(* CoDeSys 2.3 project: cy-07-wg-004.pro *)
(* Title: ClevergyAS - Albino E-02 *)
(* Version: 1.25 *)
(* Author: Andrea Ravasio *)
(* Libraries: ModbusEthernet_03.lib 20.1.16 10:42:42, Standard.lib 2.12.10 14:48:34, Util.lib 26.9.14 10:12:46, Visual.lib 2.12.10 14:48:34, LON_01.lib 28.9.12 14:05:10, WagoLibIdent.lib 25.2.13 11:12:16, WagoLibMBX_01.lib 20.3.12 16:32:40, SysLibSockets.lib 10.2.11 09:20:54, Ethernet.lib 2.12.10 14:48:32, WagoLibStatus.lib 2.12.10 14:48:32, SysLibFile.lib 2.12.10 14:48:34, SysLibRtc.lib 2.12.10 14:48:32, SysLibEvent.lib 2.12.10 14:48:34, SysLibPlcCtrl.lib 2.12.10 14:48:32, SysLibCallback.lib 2.12.10 14:48:32, Application\WagoLibEthernet_01.lib 2.12.10 14:48:36 *)

(* PLC configuration (modules and I/O channels)
VPN_ST1 AT %IX24.0 [BOOLOnX_I] Ch_1 Digital input
LAMP_AL AT %QX16.0 [BOOLOnX_Q] Ch_1 Digital output
KEY_QE_ST1 AT %IX24.1 [BOOLOnX_I] Ch_2 Digital input
CIRD05a_EN AT %QX16.1 [BOOLOnX_Q] Ch_2 Digital output
CIRD05b_AL AT %IX24.2 [BOOLOnX_I] Ch_3 Digital input
CIRD04b_EN AT %QX16.2 [BOOLOnX_Q] Ch_3 Digital output
CIRD05b_ST AT %IX24.3 [BOOLOnX_I] Ch_4 Digital input
CIRD04a_EN AT %QX16.3 [BOOLOnX_Q] Ch_4 Digital output
CIRD05b_AUT AT %IX24.4 [BOOLOnX_I] Ch_5 Digital input
CIRD03b_EN AT %QX16.4 [BOOLOnX_Q] Ch_5 Digital output
CIRD05a_AL AT %IX24.5 [BOOLOnX_I] Ch_6 Digital input
CIRD03a_EN AT %QX16.5 [BOOLOnX_Q] Ch_6 Digital output
CIRD05a_ST AT %IX24.6 [BOOLOnX_I] Ch_7 Digital input
CIRD02b_EN AT %QX16.6 [BOOLOnX_Q] Ch_7 Digital output
CIRD05a_AUT AT %IX24.7 [BOOLOnX_I] Ch_8 Digital input
CIRD02a_EN AT %QX16.7 [BOOLOnX_Q] Ch_8 Digital output
CIRD04b_AL AT %IX24.8 [BOOLOnX_I] Ch_1 Digital input
CIRD01b_EN AT %QX16.8 [BOOLOnX_Q] Ch_1 Digital output
CIRD04b_ST AT %IX24.9 [BOOLOnX_I] Ch_2 Digital input
CIRD01a_EN AT %QX16.9 [BOOLOnX_Q] Ch_2 Digital output
CIRD04b_AUT AT %IX24.10 [BOOLOnX_I] Ch_3 Digital input
CIRD05b_EN AT %QX16.10 [BOOLOnX_Q] Ch_3 Digital output
CIRD04a_AL AT %IX24.11 [BOOLOnX_I] Ch_4 Digital input
AT %QX16.11 [BOOLOnX_Q] Ch_4 Digital output
CIRD04a_ST AT %IX24.12 [BOOLOnX_I] Ch_5 Digital input
AT %QX16.12 [BOOLOnX_Q] Ch_5 Digital output
CIRD04a_AUT AT %IX24.13 [BOOLOnX_I] Ch_6 Digital input
AT %QX16.13 [BOOLOnX_Q] Ch_6 Digital output
CIRD03b_AL AT %IX24.14 [BOOLOnX_I] Ch_7 Digital input
AT %QX16.14 [BOOLOnX_Q] Ch_7 Digital output
CIRD03b_ST AT %IX24.15 [BOOLOnX_I] Ch_8 Digital input
AT %QX16.15 [BOOLOnX_Q] Ch_8 Digital output
CIRD03b_AUT AT %IX25.0 [BOOLOnX_I] Ch_1 Digital input
CIRD02b_AL AT %IX25.1 [BOOLOnX_I] Ch_2 Digital input
CIRD03a_AL AT %IX25.2 [BOOLOnX_I] Ch_3 Digital input
CIRD02b_ST AT %IX25.3 [BOOLOnX_I] Ch_4 Digital input
CIRD03a_ST AT %IX25.4 [BOOLOnX_I] Ch_5 Digital input
CIRD02b_AUT AT %IX25.5 [BOOLOnX_I] Ch_6 Digital input
CIRD03a_AUT AT %IX25.6 [BOOLOnX_I] Ch_7 Digital input
CIRD02a_AL AT %IX25.7 [BOOLOnX_I] Ch_8 Digital input
CIRD02a_ST AT %IX25.8 [BOOLOnX_I] Ch_1 Digital input
CIRD01b_AUT AT %IX25.9 [BOOLOnX_I] Ch_2 Digital input
CIRD02a_AUT AT %IX25.10 [BOOLOnX_I] Ch_3 Digital input
CIRD01a_AL AT %IX25.11 [BOOLOnX_I] Ch_4 Digital input
CIRD01b_AL AT %IX25.12 [BOOLOnX_I] Ch_5 Digital input
CIRD01a_ST AT %IX25.13 [BOOLOnX_I] Ch_6 Digital input
CIRD01b_ST AT %IX25.14 [BOOLOnX_I] Ch_7 Digital input
CIRD01a_AUT AT %IX25.15 [BOOLOnX_I] Ch_8 Digital input
ALARM_PM AT %IX26.0 [BOOLOnX_I] Ch_1 Digital input
AT %IX26.1 [BOOLOnX_I] Ch_2 Digital input
ALARM_PB AT %IX26.2 [BOOLOnX_I] Ch_3 Digital input
AT %IX26.3 [BOOLOnX_I] Ch_4 Digital input
ALARM_TB AT %IX26.4 [BOOLOnX_I] Ch_5 Digital input
AT %IX26.5 [BOOLOnX_I] Ch_6 Digital input
CTL01_ST AT %IX26.6 [BOOLOnX_I] Ch_7 Digital input
AT %IX26.7 [BOOLOnX_I] Ch_8 Digital input
AT %IB0 [BYTEOnB_I] First Byte of 24
AT %QB0 [BYTEOnB_Q] First Byte of 24
0750-0464#04 2/4 AI RTD / ADJ./ HA [Type_44_4_Channels] node 6, in %IB48 out %QB28 {INTTypePAAssignment = PLC; INTTypeModule = plugged}
  T_S01 AT %IW12 [INTOnW_I] Ch_1 signed Input value
  T_S02 AT %IW13 [INTOnW_I] Ch_2 signed Input value
  T_S03 AT %IW14 [INTOnW_I] Ch_3 signed Input value
  T_S04 AT %IW15 [INTOnW_I] Ch_4 signed Input value
0750-0464#04 2/4 AI RTD / ADJ./ HA [Type_44_4_Channels] node 7, in %IB72 out %QB52 {INTTypePAAssignment = PLC; INTTypeModule = plugged}
  T_S07 AT %IW16 [INTOnW_I] Ch_1 signed Input value
  T_S06 AT %IW17 [INTOnW_I] Ch_2 signed Input value
  T_S05 AT %IW18 [INTOnW_I] Ch_3 signed Input value
  AT %IW19 [INTOnW_I] Ch_4 signed Input value
0750-0478 2 AI 0-10V 16 Bit S.E. [Type_8_2_Channels] node 8, in %IB80 out %QB52 {INTTypePAAssignment = PLC; INTTypeModule = plugged}
  VRD01_ST AT %IW20 [WORDOnW_I] Ch_1 Input word
  VRD02_ST AT %IW21 [WORDOnW_I] Ch_2 Input word
0750-0478 2 AI 0-10V 16 Bit S.E. [Type_8_2_Channels] node 9, in %IB88 out %QB52 {INTTypePAAssignment = PLC; INTTypeModule = plugged}
  VRD03_ST AT %IW22 [WORDOnW_I] Ch_1 Input word
  AT %IW23 [WORDOnW_I] Ch_2 Input word
0750-0556 2 AO ±10V [Type_14_2_Channels] node 10, in %IB92 out %QB52 {INTTypePAAssignment = PLC; INTTypeModule = plugged}
  VRD01_CTRL AT %QW12 [WORDOnW_Q] Ch_1 Analog output
  VRD02_CTRL AT %QW13 [WORDOnW_Q] Ch_2 Analog output
0750-0556 2 AO ±10V [Type_14_2_Channels] node 11, in %IB96 out %QB52 {INTTypePAAssignment = PLC; INTTypeModule = plugged}
  VRD03_CTRL AT %QW14 [WORDOnW_Q] Ch_1 Analog output
  AT %QW15 [WORDOnW_Q] Ch_2 Analog output
Fieldbus variables [FB_VARS] node 1, in %IB0 out %QB0
Flag variables [FLAG_VARS] node 2, in %IB0 out %QB0
Modbus-Master [MB_MASTER] node 3, in %IB0 out %QB0
*)

(* Global variable list: Addiitonal_Constants *)
VAR_GLOBAL CONSTANT

	Logger_MaxBCK : WORD:=100;

END_VAR

(* Global variable list: Additional_Retain *)
VAR_GLOBAL RETAIN PERSISTENT
	LogBCKIndex:  WORD;
END_VAR

(* Global variable list: Global_Constants *)
VAR_GLOBAL CONSTANT


	Plant_NAME			: STRING :='cySN:07 cyVER: E04 Palestra Palasport Albino ';
	Plant_SN			: DWORD  :=07(*07*);	(* S/N Impianto di telecontrollo *)
	Plant_SW_VER		: WORD   :=1;		(* Versione SW installata *)


	(* Colour defines *)
	COLOR_RED			: DWORD	:= 16#2020F0;
	COLOR_YELLOW		: DWORD	:= 16#20F0F0;
	COLOR_GREEN			: DWORD	:= 16#20F020;
	COLOR_LIGHT_GREEN	: DWORD := 16#006000;

	(* Parameters *)
	Plant_DefaultTAmb	: INT	:=100;		(* [.1°C] Temperatura ambiente di default in caso di rottura sonda *)
	Plant_MaxRunTAmb	: INT   :=210; 		(* [.1°C] Temperatura ambiente massima funzionamento impianto *)
	Plant_AntiFreezeTAmb: INT   :=-40;		(* [.1°C] Antifreeze temperature, start circulators *)
	Plant_VRD_TAlarm	: INT   :=850; 		(* [.1°C] Temperatura di allarme VRD, blocco *)
	Plant_VRD_TMax		: INT   :=800; 		(* [.1°C] Setpoint massimo per uscita VRD *)
	Plant_VRD_TDefault	: INT	:=300;		(* [.1°C] Temperatura di default in caso di errore climatica *)
	Plant_CirOffDelay	: TIME	:=T#30m;	(* (Def.T#15m) Ritardo spegnimento pompe per ricircolo caldaia *)
	Plant_CirOnDelay	: TIME	:=T#15m;
	Plant_MaxWaterLoss	: WORD  :=2;		(* [lt/h] Massima perdita del circuito *)

	(* Filesystem *)
	FilesPath  			: STRING :='S:\';

	(* TCP Logger *)
	Logger_SERVER		: STRING:='';
	Logger_IP			: STRING:='192.168.100.3';(*'178.33.227.41'; (*  *) *)
	Logger_PORT			: WORD  :=80;
	Logger_GETSTART		: STRING:='GET /cygmsrv/hsgm.ashx?';
	Logger_GETEND		: STRING:='$R$N$R$N';
	Logger_CHECK		: STRING:='True';
	Logger_CRLF			: STRING:='$R$N';
	Logger_DataFile		: STRING:='S:\LOG.DAT';
	Logger_DataFileOld	: STRING:='S:\LOG.BCK';
	Logger_IndexFile	: STRING:='S:\LOG.IDX';
	Logger_ConnRetries	: BYTE:=5;
	Logger_RecoverMsgs	: BYTE:=25;

	(* TCP Remote *)
	Remote_PORT			: WORD  :=10;
	Remote_WELCOME		: STRING:='Connected$R$N';
	Remote_OK			: STRING:='OK$R$N';
	Remote_ERROR		: STRING:='ERROR$R$N';

	(* TCP Sockets *)
	MAX_SEND_TCP_SERVER					 : DWORD:=3000;(*60000*)
	MAX_RECEIVE_TCP_SERVER				 : DWORD:=3000;
	MAX_RECEIVE_TCP_SERVER_SOCKET	 	 : DWORD:=1500;
	MAX_SEND_TCP_CLIENT					 : DWORD:=3000;(*15000*)
	MAX_RECEIVE_TCP_CLIENT				 : DWORD:=1500;
	MAX_RECEIVE_TCP_CLIENT_SOCKET		 : DWORD:=1500;
	MAX_RECEIVE_UDP_SERVER				 : INT  :=1472;
	MAX_RECEIVE_UDP_CLIENT				 : INT  :=1472;
	CONNECT_WATCHDOG_TIME				 : TIME :=t#10s;

END_VAR

(* Global variable list: Global_Retain *)
VAR_GLOBAL RETAIN PERSISTENT
	CAL01_Clima : typ_Clima;
	VRD01_Clima : typ_Clima;
	VRD02_Clima : typ_Clima;
	VRD03_Clima : typ_Clima;

	CTL01_Count : DWORD;

	Mode_Manual : BOOL := FALSE;



	DelayAllarmeTemperaturaNonRaggiunta: INT;
	DeltaInterventoAllarmeTempeaturaNonRaggiuta: INT;
	OffsetSetPointManuale:INT;							(* Offset al Setpoint manuale per comensare lo scambiatore *)

	SogliaMinStartAntigelo: INT;
	SogliaMinStopAntigelo: INT;
	BitAbilitaAntigelo: BOOL:=TRUE;

END_VAR

(* Global variable list: Global_Variables *)
VAR_GLOBAL

	SYS    : typ_SYS;
	Logger : typ_Logger;


(*	Lamp	:	PLANT_STATUS; *)
	Lamp	:	LAMP_AL_GENERALE;

	T_AMB	:	INT;		(* Environment temperature *)

	TPV01  : obj_TPV	:= ( ID:=1 ); 							   (* T_S01 *)
	TPV02  : obj_TPV	:= ( ID:=2 , IN_WMIN:=50 , IN_WMAX:=870, IN_EMAX:=900 ); (* T_S02 - CAL01 - T_Send *)
	TPV03  : obj_TPV	:= ( ID:=3 , IN_WMIN:=50 , IN_WMAX:=850, IN_EMAX:=900 ); (* T_S03 *)
	TPV04  : obj_TPV	:= ( ID:=4 , IN_WMIN:=50 , IN_WMAX:=800 ); (* T_S04 *)
	TPV05  : obj_TPV	:= ( ID:=5 , IN_WMIN:=50 , IN_WMAX:=800 ); (* T_S05 *)
	TPV06  : obj_TPV	:= ( ID:=6 , IN_WMIN:=50 , IN_WMAX:=800 ); (* T_S06 *)
	TPV07  : obj_TPV	:= ( ID:=7 , IN_WMIN:=50 , IN_WMAX:=800 ); (* T_S07 *)
	TPV08  : obj_TPV	:= ( ID:=8 , IN_WMIN:=50 , IN_WMAX:=800 ); (* T_S08 per Gestione SPLIT *)
	TPV09  : obj_TPV	:= ( ID:=9 , IN_WMIN:=50 , IN_WMAX:=800 ); (* T_S09 per Gestione SPLIT *)
	TPV10  : obj_TPV	:= ( ID:=10 , IN_WMIN:=50 , IN_WMAX:=800 ); (* T_S10 per Gestione SPLIT *)
	TPV11  : obj_TPV	:= ( ID:=11 , IN_WMIN:=50 , IN_WMAX:=800 ); (* T_S11 per Gestione SPLIT *)

	TAMB   : obj_TAMB	:= ( ID:=1 );

	CAL01  : obj_CAL_VT100GC1B := ( ID:=1 );

	THER01 : obj_CRONTER_01 := ( ID:=1, Local_MaxRunTAmb:=250,Histeresys:=10);  (* Controllo Split 10 e 11 *)
	THER02 : obj_CRONTER_01 := ( ID:=2, Local_MaxRunTAmb:=250,Histeresys:=10);	(* Controllo SPLIt 4,5 e 6 *)
	THER03 : obj_CRONTER_01 := ( ID:=3, Local_MaxRunTAmb:=250,Histeresys:=10);	(* Controllo Split 8,9 e 10 *)
	THER04 : obj_CRONTER_01 := ( ID:=4, Local_MaxRunTAmb:=250,Histeresys:=10);	(* Controllo SPLIt 1,2 e 3 *)
	THER05 : obj_CRONTER_01 := ( ID:=5, Local_MaxRunTAmb:=250,Histeresys:=10);	(* Controllo Circolatore CIRD05 Servizi *)
	THER06 : obj_CRONTER_01 := ( ID:=6, Local_MaxRunTAmb:=800,Histeresys:=10);	(* Controllo Circolatore CIRD02 Bollitore *)
	THER07 : obj_CRONTER_01 := ( ID:=7, Local_MaxRunTAmb:=250,Histeresys:=10);	(* Controllo Ciroclatore CIRD03 ACS *)
	THER250 : obj_CRONTER_01 := ( ID:=250 );	(* Controllo Boost *)

	CronEd : obj_CRON_EDITOR_01;

	(* Circolatori  *)
	CIRD01 :obj_CIR_DOPPIO_new := (ID:=1, OnDelay:=T#1m, ExtStatus:=FALSE, Mode:=1); (* Primario Caldaia *)
	CIRD02 :obj_CIR_DOPPIO_new := (ID:=2, OnDelay:=T#1m, ExtStatus:=FALSE, Mode:=0); (* Secondario Bollitore *)
	CIRD03 :obj_CIR_DOPPIO_new := (ID:=3, OnDelay:=T#1m, ExtStatus:=FALSE, Mode:=0); (* Secondario ACS *)
	CIRD04 :obj_CIR_DOPPIO_new := (ID:=4, OnDelay:=T#1m, ExtStatus:=FALSE, Mode:=0); (* Secondario Ariotermi *)
	CIRD05 :obj_CIR_DOPPIO_new := (ID:=5, OnDelay:=T#1m, ExtStatus:=FALSE, Mode:=0); (* Secondario Servizi *)



	(* Valvole motorizzate Analogiche  *)
	VRD01	:	obj_VRD_new	:= (ID:=1, fFeedback:=TRUE, ReducedRange := FALSE , Local_VRD_TAlarm:=800);
	VRD02	:	obj_VRD_new := (ID:=2, fFeedback:=TRUE, ReducedRange := FALSE , Local_VRD_TAlarm:=800);
	VRD03	:	obj_VRD_new := (ID:=3, fFeedback:=TRUE, ReducedRange := FALSE, Local_VRD_TAlarm:=800);

	CTL01	:	obj_CTL	:= (ID:=1, Peso:=100);  (**** 0,5 litri al minuto : 2 impulsi al litro ***)

	SPL01:obj_SPLIT:= ( ID:=1);
	SPL02:obj_SPLIT:= ( ID:=2);
	SPL03:obj_SPLIT:= ( ID:=3);
	SPL04:obj_SPLIT:= ( ID:=4);
	SPL05:obj_SPLIT:= ( ID:=5);
	SPL06:obj_SPLIT:= ( ID:=6);
	SPL07:obj_SPLIT:= ( ID:=7);
	SPL08:obj_SPLIT:= ( ID:=8);
	SPL09:obj_SPLIT:= ( ID:=9);
	SPL10:obj_SPLIT:= ( ID:=10);
	SPL11:obj_SPLIT:= ( ID:=11);


(* Variabili Globali letti dal remoto della Palestra *)

	KEY_QE_ST2: BOOL;
	SPLIT06_ST: BOOL;
	SPLIT08_ST: BOOL;
	SPLIT05_ST: BOOL;
	SPLIT07_ST: BOOL;
	SPLIT04_ST: BOOL;
	SPLIT01_ST: BOOL;
	SPLIT09_ST: BOOL;
	SPLIT02_ST: BOOL;
	SPLIT11_ST: BOOL;
	SPLIT03_ST: BOOL;
	SPLIT10_ST: BOOL;
	SPLIT06_EN: BOOL;
	SPLIT05_EN: BOOL;
	SPLIT04_EN: BOOL;
	SPLIT09_EN: BOOL;
	SPLIT08_EN: BOOL;
	SPLIT07_EN: BOOL;
	SPLIT01_EN: BOOL;
	SPLIT02_EN: BOOL;
	SPLIT03_EN: BOOL;
	SPLIT11_EN: BOOL;
	SPLIT10_EN: BOOL;


	T_S08:INT;
	T_S09:INT;
	T_S10:INT;
	T_S11:INT;







END_VAR

(* Global variable list: LON/Module_1/InterfaceBlock_Module_1 *)
VAR_GLOBAL CONSTANT
(******************************************)
(* Automatic generated code, do not edit! *)
(******************************************)
	abSignature_Module_1 : ARRAY[0..15] OF BYTE := 16#B4,16#A9,16#CB,16#FD,16#2D,16#5A,16#D7,16#4A,16#B1,16#7E,16#A8,16#70,16#0A,16#0F,16#B9,16#03;
	wConfigSize_Module_1 : WORD := 421;
	abInterface_Module_1 : ARRAY[0..105] OF DWORD :=
		16#50A640DC, 16#219F340B, 16#6041B800, 16#06246830, 16#428B2E71, 16#64B95263, 16#FE000902, 16#2A050140, 
		16#0028408B, 16#20280AF2, 16#80A205C4, 16#685174C0, 16#8E03020C, 16#B8AB63AE, 16#953A4EEA, 16#AA63AD8E, 
		16#63ACD182, 16#4EEB98AD, 16#313DBE3A, 16#A6020F80, 16#13011245, 16#9926B18A, 16#0994A6CB, 16#508D4E85, 
		16#F6AD5BAA, 16#C53E2D4B, 16#EED8B26A, 16#920DBA93, 16#DBBC20C9, 16#0529B7EE, 16#B66DDF8E, 16#49D76DD9, 
		16#72CBA205, 16#1626C0B2, 16#A5A6B5EB, 16#6CDDB865, 16#4CA03BB7, 16#8AC91726, 16#3BF5AD0C, 16#75E986A5, 
		16#E2C9A3B9, 16#5AA34208, 16#4054966D, 16#946ACAA7, 16#49264935, 16#23655360, 16#E3E92DD4, 16#1524C09B, 
		16#A97EA56A, 16#4E053D69, 16#C906C1CA, 16#54CA1922, 16#E586651B, 16#12B5706D, 16#D3AF5791, 16#A0FA824C, 
		16#D202B450, 16#D069007C, 16#A940D4E8, 16#EAC16D51, 16#83B21003, 16#8B579930, 16#79D912B9, 16#02ED1029, 
		16#DDB14145, 16#6D5B962A, 16#B7471BC0, 16#511C9520, 16#3D44BB68, 16#1BAC9C4E, 16#61E7861D, 16#A1D85F80, 
		16#823280B0, 16#B3FF0007, 16#6C109AC5, 16#30A13C03, 16#E2386308, 16#58DB08B0, 16#6F400DE6, 16#0701DA1C, 
		16#98F51C73, 16#40A0630F, 16#AEE3AF23, 16#632020C0, 16#402040AF, 16#1605B0E3, 16#185B0CC4, 16#EDC04D71, 
		16#0610584B, 16#001688C7, 16#4544F1F8, 16#1C1713C6, 16#71815C54, 16#CA454672, 16#0696150F, 16#120412D0, 
		16#4C973101, 16#44A16C67, 16#2820D488, 16#E04081E0, 16#2F4F4D9B, 16#75AD2DFB, 16#F61B5BE9, 16#870AE1A2, 
		16#1B7860EE, 16#00000090;
END_VAR

(* Global variable list: LON/Module_1/Runtime_Module_1 *)
VAR_GLOBAL
(******************************************)
(* Automatic generated code, do not edit! *)
(******************************************)
	mbxModule_1 : MBX_Full;
	InDataTelegram_Module_1 : ARRAY[0..255] OF BYTE;
	OutDataTelegram_Module_1 : ARRAY[0..511] OF BYTE;

	xInitRunning_Module_1 : BOOL := FALSE;
	unLastLen_mbxModule_1 : UINT;
END_VAR

(* Data type in LON/Enumerations *)
TYPE alarm_type_t :
(
	AL_HEADER := -13,
	AL_FOOTER := -12,
	AL_DEBUG := -11,
	AL_INFO := -10,
	AL_SYSTEM_INFO := -6,
	AL_VALUE_INVALID := -5,
	AL_CONSTANT := -4,
	AL_OFFLINE := -3,
	AL_UNKNOWN := -2,
	AL_NUL := -1,
	AL_NO_CONDITION := 0,
	AL_ALM_CONDITION := 1,
	AL_TOT_SVC_ALM_1 := 2,
	AL_TOT_SVC_ALM_2 := 3,
	AL_TOT_SVC_ALM_3 := 4,
	AL_LOW_LMT_CLR_1 := 5,
	AL_LOW_LMT_CLR_2 := 6,
	AL_HIGH_LMT_CLR_1 := 7,
	AL_HIGH_LMT_CLR_2 := 8,
	AL_LOW_LMT_ALM_1 := 9,
	AL_LOW_LMT_ALM_2 := 10,
	AL_HIGH_LMT_ALM_1 := 11,
	AL_HIGH_LMT_ALM_2 := 12,
	AL_FIR_ALM := 13,
	AL_FIR_PRE_ALM := 14,
	AL_FIR_TRBL := 15,
	AL_FIR_SUPV := 16,
	AL_FIR_TEST_ALM := 17,
	AL_FIR_TEST_PRE_ALM := 18,
	AL_FIR_ENVCOMP_MAX := 19,
	AL_FIR_MONITOR_COND := 20,
	AL_FIR_MAINT_ALERT := 21,
	AL_FATAL_ERROR := 30,
	AL_ERROR := 31,
	AL_WARNING := 32
);
END_TYPE

(* Data type in Errors *)
TYPE en_Logger_ErrLev :
(
	EL_Log			:=0,
	EL_Wrn			:=1,
	EL_Alarm		:=2,
	EL_AlarmStop	:=3
);
END_TYPE

(* Data type in Errors *)
TYPE en_Logger_Status :
(
	S_Logger_UNKNOWN := 0,
	S_Logger_IDLE,
	S_Logger_WAITCONN,
	S_Logger_WAITTX,
	S_Logger_WAITRESP,
	S_Logger_ERROR
);
END_TYPE

(* Data type *)
TYPE en_SYS_Objects :
(
	EO_SYS		:=0,  (* PLC *)
	EO_VPN		:=1,  (* VPN *)
	EO_DOOR		:=2,  (* Door & access control *)

	EO_CAL		:=10, (* Caldaia *)
	EO_CIR		:=11, (* Circolatore *)
	EO_CRON		:=12, (* Crono-termostato *)
	EO_VRD		:=13, (* Valvola miscelatore pannelli *)
	EO_CTL		:=14, (* Contalitri *)
	EO_CTB		:=15, (* Contabilizzatore *)
	EO_TPV		:=16, (* Temperature probes values *)
	EO_PPV		:=17, (* Pressure probes values *)
	EO_PBV		:=18, (* Over-Pressure Alarms *)
	EO_TBV		:=19, (* Over-Temperature Alarms *)
	EO_PMV		:=20, (* Under-Pressure Alarms *)
	EO_GRU		:=21, (* Gruppo termico *)
	EO_PDC		:=22, (* Pompa di calore *)
	EO_SOL		:=23, (* Pannello solare termico *)
	EO_ESOL		:=24, (* Pannello solare fotovoltaico *)
	EO_GAS		:=25, (* Contatore GAS *)
	EO_PORT		:=26, (* Misuratore di portata *)
	EO_FPV		:=27, (* Flow probes values *)
	EO_ANZ		:=28, (* Analizzatore di rete *)
	EO_SCA		:=29, (* Signal Control Alarms *)
	EO_LUX		:=30, (* Base Illumination point *)
	EO_LUXM		:=31, (* Metered Illumination point *)
	EO_PSG		:=32, (* Sensore di passaggio *)
	EO_HVAC		:=33, (* Heating, Ventilating and Air Conditioning *)
	EO_HYGRV	:=34, (* Relative Humidity sensors value *)
	EO_COOV		:=35, (* Carbon Dioxide CO2 sensors value *)
	EO_INV		:=36, (* Inverter *)
	EO_STR		:=37, (* Smart string box *)

	EO_SPT		:=38, (* SPLIT *)

	EO_CIRD		:=39, (* Double CIR *)
	EO_ACS		:=40, (* Hot domestic water *)
	EO_FRG		:=41, (* Frigo *)
	EO_THER		:=42, (* Thermostat *)
	EO_CIRM		:=43, (* Modbus CIR *)
	EO_CIRDM	:=44, (* Modbus double CIR *)

	EO_ZGW			:=200,  (* ZigBee - Gateway *)
	EO_ZRM			:=201,	(* ZigBee - Repeater *)
	EO_ZREL			:=202,	(* ZigBee - Actuator rele *)
	EO_ZTHL			:=203,	(* ZigBee - Temperature Sensor *)

	EO_ASGW			:=250,	(* ASi - Gateway *)
	EO_ASCBI		:=251,	(* ASi - Input Board, Ciabatta *)

	EO_LON			:=1000, (* Bus - LON *)
	EO_MODBUS		:=1001, (* Bus - MODBUS *)
	EO_MBUS			:=1002, (* Bus - M-BUS *)
	EO_MODBUS_TCP	:=1003, (* Bus - MODBUS TCP *)

	EO_GENERIC		:=9000, (* Generic dataset *)
	EO_EXPO			:=9001 (* EXPO dataset *)
);
END_TYPE

(* Data type *)
TYPE en_SYS_Status :
(
	S_UNKNOWN  := 0,
	S_STARTUP,
	S_INIT_RTC,
	S_INIT_VAR,
	S_AUTOTEST,
	S_RUNNING,
	S_SHUTDOWN,
	S_HALT
);
END_TYPE

(* Data type in LON/Enumerations *)
TYPE file_request_t :
(
	FR_NUL := -1,
	FR_OPEN_TO_SEND := 0,
	FR_OPEN_TO_RECEIVE := 1,
	FR_CLOSE_FILE := 2,
	FR_CLOSE_DELETE_FILE := 3,
	FR_DIRECTORY_LOOKUP := 4,
	FR_OPEN_TO_SEND_RA := 5,
	FR_OPEN_TO_RECEIVE_RA := 6
);
END_TYPE

(* Data type in LON/Enumerations *)
TYPE file_status_t :
(
	FS_NUL := -1,
	FS_XFER_OK := 0,
	FS_LOOKUP_OK := 1,
	FS_OPEN_FAIL := 2,
	FS_LOOKUP_ERR := 3,
	FS_XFER_UNDERWAY := 4,
	FS_IO_ERR := 5,
	FS_TIMEOUT_ERR := 6,
	FS_WINDOW_ERR := 7,
	FS_AUTH_ERR := 8,
	FS_ACCESS_UNAVAIL := 9,
	FS_SEEK_INVALID := 10,
	FS_SEEK_WAIT := 11
);
END_TYPE

(* Data type in LON/Enumerations *)
TYPE hvac_t :
(
	HVAC_NUL := -1,
	HVAC_AUTO := 0,
	HVAC_HEAT := 1,
	HVAC_MRNG_WRMUP := 2,
	HVAC_COOL := 3,
	HVAC_NIGHT_PURGE := 4,
	HVAC_PRE_COOL := 5,
	HVAC_OFF := 6,
	HVAC_TEST := 7,
	HVAC_EMERG_HEAT := 8,
	HVAC_FAN_ONLY := 9,
	HVAC_FREE_COOL := 10,
	HVAC_ICE := 11,
	HVAC_MAX_HEAT := 12,
	HVAC_ECONOMY := 13,
	HVAC_DEHUMID := 14,
	HVAC_CALIBRATE := 15,
	HVAC_EMERG_COOL := 16,
	HVAC_EMERG_STEAM := 17,
	HVAC_MAX_COOL := 18,
	HVAC_HVC_LOAD := 19,
	HVAC_NO_LOAD := 20
);
END_TYPE

(* Data type in LON/Enumerations *)
TYPE object_request_t :
(
	RQ_NUL := -1,
	RQ_NORMAL := 0,
	RQ_DISABLED := 1,
	RQ_UPDATE_STATUS := 2,
	RQ_SELF_TEST := 3,
	RQ_UPDATE_ALARM := 4,
	RQ_REPORT_MASK := 5,
	RQ_OVERRIDE := 6,
	RQ_ENABLE := 7,
	RQ_RMV_OVERRIDE := 8,
	RQ_CLEAR_STATUS := 9,
	RQ_CLEAR_ALARM := 10,
	RQ_ALARM_NOTIFY_ENABLED := 11,
	RQ_ALARM_NOTIFY_DISABLED := 12,
	RQ_MANUAL_CTRL := 13,
	RQ_REMOTE_CTRL := 14,
	RQ_PROGRAM := 15,
	RQ_CLEAR_RESET := 16,
	RQ_RESET := 17,
	RQ_CLEAR_LOG := 18,
	RQ_LOAD_PROGRAM := 19,
	RQ_RUN_PROGRAM := 20,
	RQ_HALT_PROGRAM := 21,
	RQ_RESTART_PROGRAM := 22,
	RQ_UNLOAD_PROGRAM := 23,
	RQ_STEP_PROGRAM := 24
);
END_TYPE

(* Data type in LON/Enumerations *)
TYPE priority_level_t :
(
	PR_NUL := -1,
	PR_LEVEL_0 := 0,
	PR_LEVEL_1 := 1,
	PR_LEVEL_2 := 2,
	PR_LEVEL_3 := 3,
	PR_1 := 4,
	PR_2 := 5,
	PR_3 := 6,
	PR_4 := 7,
	PR_6 := 8,
	PR_8 := 9,
	PR_10 := 10,
	PR_16 := 11
);
END_TYPE

(* Data type in Plant_Objects *)
TYPE typ_Clima : (* CURVA CLIMATICA *)
STRUCT
	InitOK:		BOOL;
	Points: 	ARRAY [0..10] OF POINT;
END_STRUCT
END_TYPE

(* Data type in Plant_Objects *)
TYPE typ_Cron_Calendar :
STRUCT
	Profile		: ARRAY[0..384] OF BYTE;
END_STRUCT
END_TYPE

(* Data type in Plant_Objects *)
TYPE typ_Cron_Jolly :
STRUCT
	Start		: DT;
	End			: DT;
	Temp		: WORD;
	Flags		: WORD; (* B0:Enabled B1..B15:Unused *)
END_STRUCT
END_TYPE

(* Data type in Plant_Objects *)
TYPE typ_Cron_Profile :
STRUCT
	Flags		: WORD;
	Setpoint	: ARRAY [0..95] OF WORD;
END_STRUCT
END_TYPE

(* Data type in Errors *)
TYPE typ_Logger :
STRUCT
	Status		: en_Logger_Status;

	SendReq		: BOOL;
	SendIdx		: DWORD;
	SendData	: ARRAY [0..MAX_SEND_TCP_CLIENT] OF BYTE;
	SendLen		: DINT;

	TData		: ARRAY [0..MAX_SEND_TCP_CLIENT] OF BYTE;
	TLen		: DINT;

	LastIdxPos	: DWORD;

	(* Temporary variables used by objects *)
	s1			: STRING(256);
	i1			: WORD;

END_STRUCT
END_TYPE

(* Data type in Plant_Objects *)
TYPE typ_MODBUS_VAR : (* Gestione parametri MODBUS *)
STRUCT
	SlaveAddress	: BYTE;
	FunCode			: BYTE;
	FunAddress		: WORD;
	Refresh_Time	: BYTE; (* 0:No refresh x:Refresh in seconds *)
	Refresh_Cnt		: BYTE; (* INTERNAL *)
	Variable		: POINTER TO WORD;
	Variable_Size	: BYTE;
	Variable_Mirror : WORD; (* INTERNAL [Force refresh on read variables when <>0] *)
END_STRUCT
END_TYPE

(* Data type *)
TYPE typ_SYS :
STRUCT
	Status			: en_SYS_Status;
	Warning			: BOOL;
	Alarm			: BOOL;
	AlarmStop		: BOOL;

	Time_LogString	: STRING;
	Time_Year		: WORD;
	Time_Month		: BYTE;
	Time_Day		: BYTE;
	Time_Hour		: BYTE;
	Time_Minute		: BYTE;

	Time_CT_DT		: DT;
	Time_CT_Day		: WORD;
	Time_CT_Quarter	: BYTE;

	LastLogs_Idx	: BYTE;
	LastLogs_Dat	: ARRAY[0..5] OF STRING;
	LastLogs_Msg	: ARRAY[0..5] OF STRING;

END_STRUCT
END_TYPE

(* Data type in LON/NetworkVariables *)
TYPE typSnvtAlarm : 
STRUCT
	abLocation : ARRAY[0..5] OF BYTE;
	wObjectId : WORD;
	bAlarmType : BYTE (* enum type alarm_type_t *);
	bPriorityLevel : BYTE (* enum type priority_level_t *);
	wIndexToSnvt : WORD;
	abValue : ARRAY[0..3] OF BYTE;
	wYear : WORD;
	bMonth : BYTE;
	bDay : BYTE;
	bHour : BYTE;
	bMinute : BYTE;
	bSecond : BYTE;
	wMillisecond : WORD;
	abAlarmLimit : ARRAY[0..3] OF BYTE;
	bStatusInformation : BYTE; (* bit allocation of bStatusInformation:
	bit 0: NVI update counter LSB
	bit 1: NVI update counter
	bit 2: NVI update counter
	bit 3: NVI update counter MSB
	bit 4: timeout for NVI occurs (MaxRcvTime expired)
	bit 5: reserved
	bit 6: reserved
	bit 7: force NVO update *)
	bInternalUseOnly : BYTE; (* Do not use this byte in your application! *)
END_STRUCT
END_TYPE

(* Data type in LON/NetworkVariables *)
TYPE typSnvtFilePos : 
STRUCT
	diRwPtr : DINT;
	wRwLength : WORD;
	bStatusInformation : BYTE; (* bit allocation of bStatusInformation:
	bit 0: NVI update counter LSB
	bit 1: NVI update counter
	bit 2: NVI update counter
	bit 3: NVI update counter MSB
	bit 4: timeout for NVI occurs (MaxRcvTime expired)
	bit 5: reserved
	bit 6: reserved
	bit 7: force NVO update *)
	bInternalUseOnly : BYTE; (* Do not use this byte in your application! *)
END_STRUCT
END_TYPE

(* Data type in LON/NetworkVariables *)
TYPE typSnvtFileReq : 
STRUCT
	bRequest : BYTE (* enum type file_request_t *);
	wIndex : WORD;
	wReceiveTimeout : WORD;
	abDestAddress : ARRAY[0..4] OF BYTE (* union declaration *);
	bAuthOn : BYTE;
	bPrioOn : BYTE;
	bStatusInformation : BYTE; (* bit allocation of bStatusInformation:
	bit 0: NVI update counter LSB
	bit 1: NVI update counter
	bit 2: NVI update counter
	bit 3: NVI update counter MSB
	bit 4: timeout for NVI occurs (MaxRcvTime expired)
	bit 5: reserved
	bit 6: reserved
	bit 7: force NVO update *)
	bInternalUseOnly : BYTE; (* Do not use this byte in your application! *)
END_STRUCT
END_TYPE

(* Data type in LON/NetworkVariables *)
TYPE typSnvtFileStatus : 
STRUCT
	bStatus : BYTE (* enum type file_status_t *);
	wNumberOfFiles : WORD;
	wSelectedFile : WORD;
	abAdr : ARRAY[0..21] OF BYTE (* union declaration *);
	bStatusInformation : BYTE; (* bit allocation of bStatusInformation:
	bit 0: NVI update counter LSB
	bit 1: NVI update counter
	bit 2: NVI update counter
	bit 3: NVI update counter MSB
	bit 4: timeout for NVI occurs (MaxRcvTime expired)
	bit 5: reserved
	bit 6: reserved
	bit 7: force NVO update *)
	bInternalUseOnly : BYTE; (* Do not use this byte in your application! *)
END_STRUCT
END_TYPE

(* Data type in LON/NetworkVariables *)
TYPE typSnvtHvacMode : 
STRUCT
	bSnvtHvacMode : BYTE (* enum type hvac_t *);
	bStatusInformation : BYTE; (* bit allocation of bStatusInformation:
	bit 0: NVI update counter LSB
	bit 1: NVI update counter
	bit 2: NVI update counter
	bit 3: NVI update counter MSB
	bit 4: timeout for NVI occurs (MaxRcvTime expired)
	bit 5: reserved
	bit 6: reserved
	bit 7: force NVO update *)
	bInternalUseOnly : BYTE; (* Do not use this byte in your application! *)
END_STRUCT
END_TYPE

(* Data type in LON/NetworkVariables *)
TYPE typSnvtObjRequest : 
STRUCT
	wObjectId : WORD;
	bObjectRequest : BYTE (* enum type object_request_t *);
	bStatusInformation : BYTE; (* bit allocation of bStatusInformation:
	bit 0: NVI update counter LSB
	bit 1: NVI update counter
	bit 2: NVI update counter
	bit 3: NVI update counter MSB
	bit 4: timeout for NVI occurs (MaxRcvTime expired)
	bit 5: reserved
	bit 6: reserved
	bit 7: force NVO update *)
	bInternalUseOnly : BYTE; (* Do not use this byte in your application! *)
END_STRUCT
END_TYPE

(* Data type in LON/NetworkVariables *)
TYPE typSnvtObjStatus : 
STRUCT
	wObjectId : WORD;
	bBitfieldByteOffset2 : BYTE (* bit field *);
	bBitfieldByteOffset3 : BYTE (* bit field *);
	bBitfieldByteOffset4 : BYTE (* bit field *);
	bBitfieldByteOffset5 : BYTE (* bit field *);
	bStatusInformation : BYTE; (* bit allocation of bStatusInformation:
	bit 0: NVI update counter LSB
	bit 1: NVI update counter
	bit 2: NVI update counter
	bit 3: NVI update counter MSB
	bit 4: timeout for NVI occurs (MaxRcvTime expired)
	bit 5: reserved
	bit 6: reserved
	bit 7: force NVO update *)
	bInternalUseOnly : BYTE; (* Do not use this byte in your application! *)
END_STRUCT
END_TYPE

(* Data type in LON/NetworkVariables *)
TYPE typSnvtState : 
STRUCT
	bBitfieldByteOffset0 : BYTE (* bit field *);
	bBitfieldByteOffset1 : BYTE (* bit field *);
	bStatusInformation : BYTE; (* bit allocation of bStatusInformation:
	bit 0: NVI update counter LSB
	bit 1: NVI update counter
	bit 2: NVI update counter
	bit 3: NVI update counter MSB
	bit 4: timeout for NVI occurs (MaxRcvTime expired)
	bit 5: reserved
	bit 6: reserved
	bit 7: force NVO update *)
	bInternalUseOnly : BYTE; (* Do not use this byte in your application! *)
END_STRUCT
END_TYPE

(* Data type in LON/NetworkVariables *)
TYPE typSnvtSwitch : 
STRUCT
	bValue : BYTE;
	siState : SINT;
	bStatusInformation : BYTE; (* bit allocation of bStatusInformation:
	bit 0: NVI update counter LSB
	bit 1: NVI update counter
	bit 2: NVI update counter
	bit 3: NVI update counter MSB
	bit 4: timeout for NVI occurs (MaxRcvTime expired)
	bit 5: reserved
	bit 6: reserved
	bit 7: force NVO update *)
	bInternalUseOnly : BYTE; (* Do not use this byte in your application! *)
END_STRUCT
END_TYPE

(* Data type in LON/NetworkVariables *)
TYPE typSnvtTempP : 
STRUCT
	iSnvtTempP : INT;
	bStatusInformation : BYTE; (* bit allocation of bStatusInformation:
	bit 0: NVI update counter LSB
	bit 1: NVI update counter
	bit 2: NVI update counter
	bit 3: NVI update counter MSB
	bit 4: timeout for NVI occurs (MaxRcvTime expired)
	bit 5: reserved
	bit 6: reserved
	bit 7: force NVO update *)
	bInternalUseOnly : BYTE; (* Do not use this byte in your application! *)
END_STRUCT
END_TYPE

(* Data type in LON/NetworkVariables *)
TYPE typSnvtTimeStamp : 
STRUCT
	iYear : INT;
	bMonth : BYTE;
	bDay : BYTE;
	bHour : BYTE;
	bMinute : BYTE;
	bSecond : BYTE;
	bStatusInformation : BYTE; (* bit allocation of bStatusInformation:
	bit 0: NVI update counter LSB
	bit 1: NVI update counter
	bit 2: NVI update counter
	bit 3: NVI update counter MSB
	bit 4: timeout for NVI occurs (MaxRcvTime expired)
	bit 5: reserved
	bit 6: reserved
	bit 7: force NVO update *)
	bInternalUseOnly : BYTE; (* Do not use this byte in your application! *)
END_STRUCT
END_TYPE

(* POU PLC_PRG, ST *)
PROGRAM PLC_PRG
VAR
	Timer1: TON; (* Fast controls tick *)
	Timer2: TON; (* Plant control tick *)
	Timer3: TON; (* Logger timer *)

(* Comunizaione con nodo WAGO 192.168.100.4 *)


	Master_1				:	ETHERNET_MODBUSMASTER_UDP;
	Funktion				:	BYTE := 16#17; 				(* READ_WRITE_REGISTERS *)

	ReadAddress				:	WORD := 16#0000;			(* Startadresse 		*)
	ReadQuantity			:	WORD := 16#0005;			(* Anzahl der Worte 	*)
	Rec_Buffer				:	ARRAY[1..255] OF WORD;	(* Empfangsdaten 	*)

	WriteAddress			:	WORD := 16#0000;			(* Startadresse		*)
	WriteQuantity			:	WORD := 16#0001;			(* Anzahl der Worte	*)
	Send_Buffer			:	ARRAY[1..255] OF WORD;	(* Sendedaten			*)

	Fehler					:	WORD;
	Fertig					:	BOOL;
	T1						:	TON;
	Z1						:	CTU;

	WordAppoggio: WORD;
	DelayAvvioCollegamentoWAGO: TON;
	HMI_AggiornaLog: BOOL;
	DelayAggiornamento: TON;
	TrigR_THER01: F_TRIG;
	VarApp: INT;
END_VAR



VAR_INPUT
	WriteOUT: WORD;
END_VAR

VAR_OUTPUT
	ReadWord: WORD;
END_VAR
(******************************************************************************
 ****                           MAIN TASK CODE                             ****
 ******************************************************************************

	Network setup:
		IP  = 192.168.100.2 | MSK = 255.255.255.0
		GW	= 192.168.100.1 | DNS = 192.168.100.1
		SNTP = 193.204.114.232 (3600s) ==> 192.168.100.3
*)

(*==============================*)
(*===== Main status machine ====*)
(*==============================*)
Main_Stm();



WordAppoggio.0:=SPLIT07_EN;
WordAppoggio.1:=SPLIT08_EN;
WordAppoggio.2:=SPLIT09_EN;
WordAppoggio.3:=SPLIT03_EN;
WordAppoggio.4:=SPLIT02_EN;
WordAppoggio.5:=SPLIT01_EN;
WordAppoggio.6:=SPLIT06_EN;
WordAppoggio.7:=SPLIT05_EN;
WordAppoggio.8:=SPLIT04_EN;
WordAppoggio.9:=SPLIT10_EN;
WordAppoggio.10:=SPLIT11_EN;
WriteOUT:=WordAppoggio;

DelayAvvioCollegamentoWAGO(IN:=TRUE , PT:=t#10s , Q=> , ET=> );
(* Provo a ritardare la lettura del nodo per veririfcare se il download del programma è più veloce *)
DelayAggiornamento(IN:=NOT DelayAggiornamento.Q,pt:=t#1s);

Fertig:=DelayAvvioCollegamentoWAGO.Q AND DelayAggiornamento.Q;

NodoWAGO();

KEY_QE_ST2:=ReadWord.0;
SPLIT03_ST:=ReadWord.1;
SPLIT07_ST:=ReadWord.2;
SPLIT02_ST:=ReadWord.3;
SPLIT08_ST:=ReadWord.4;
SPLIT01_ST:=ReadWord.5;
SPLIT09_ST:=ReadWord.6;
SPLIT06_ST:=ReadWord.7;
SPLIT05_ST:=ReadWord.8;
SPLIT10_ST:=ReadWord.9;
SPLIT04_ST:=ReadWord.10;
SPLIT11_ST:=ReadWord.11;



(*==============================*)
(*== Running cycle operations ==*)
(*==============================*)
IF SYS.Status>S_INIT_VAR THEN

	(* Update LON output variables (needs to be here to obtain only one refresh) *)
	CAL01.Heartbeat( CLIM:=CAL01_Clima );

	(* Execute LON process *)
	Module_1_PRG();

	(* Count water pulses *)
	CTL01(CTL_ST:=CTL01_ST, COUNT:=CTL01_Count);

			CIRD01(
					PumpA_AUTO:=CIRD01a_AUT,
					PumpB_AUTO:=CIRD01b_AUT ,
					PumpA_En=>CIRD01a_EN ,
					PumpB_EN=>CIRD01b_EN ,
					PumpA_AL:=NOT CIRD01a_AL,
					PumpB_AL:=NOT CIRD01b_AL,
					PumpA_ST:=CIRD01a_ST ,
					PumpB_ST:=CIRD01b_ST );

			CIRD02(
					PumpA_AUTO:=CIRD02a_AUT,
					PumpB_AUTO:=CIRD02b_AUT ,
					PumpA_En=>CIRD02a_EN ,
					PumpB_EN=>CIRD02b_EN ,
					PumpA_AL:=NOT CIRD02a_AL,
					PumpB_AL:=NOT CIRD02b_AL,
					PumpA_ST:=CIRD02a_ST ,
					PumpB_ST:=CIRD02b_ST );


			CIRD03(
					PumpA_AUTO:=CIRD03a_AUT,
					PumpB_AUTO:=CIRD03b_AUT ,
					PumpA_En=>CIRD03a_EN ,
					PumpB_EN=>CIRD03b_EN ,
					PumpA_AL:=NOT CIRD03a_AL,
					PumpB_AL:=NOT CIRD03b_AL,
					PumpA_ST:=CIRD03a_ST ,
					PumpB_ST:=CIRD03b_ST );

			CIRD04(
					PumpA_AUTO:=CIRD04a_AUT,
					PumpB_AUTO:=TRUE, (*CIRD04b_AUT , *)  (* questo ciroclatore è automatico *)
					PumpA_En=>CIRD04a_EN ,
					PumpB_EN=>CIRD04b_EN ,
					PumpA_AL:=NOT CIRD04a_AL,
					PumpB_AL:=NOT CIRD04b_AL,
					PumpA_ST:=CIRD04a_ST ,
					PumpB_ST:=CIRD04b_ST );

			CIRD05(
					PumpA_AUTO:=CIRD05a_AUT,
					PumpB_AUTO:=CIRD05b_AUT ,
					PumpA_En=>CIRD05a_EN ,
					PumpB_EN=>CIRD05b_EN ,
					PumpA_AL:=NOT CIRD05a_AL,
					PumpB_AL:=NOT CIRD05b_AL,
					PumpA_ST:=CIRD05a_ST ,
					PumpB_ST:=CIRD05b_ST );

(* SPLIT *)


			SPL01(	FeedBack_Contatore:=SPLIT01_ST ,SSPLIT_EN=> SPLIT01_EN );
			SPL02(	FeedBack_Contatore:=SPLIT02_ST ,SSPLIT_EN=> SPLIT02_EN );
			SPL03(	FeedBack_Contatore:=SPLIT03_ST ,SSPLIT_EN=> SPLIT03_EN );

			SPL04(	FeedBack_Contatore:=SPLIT04_ST ,SSPLIT_EN=> SPLIT04_EN );
			SPL05(	FeedBack_Contatore:=SPLIT05_ST ,SSPLIT_EN=> SPLIT05_EN );
			SPL06(	FeedBack_Contatore:=SPLIT06_ST ,SSPLIT_EN=> SPLIT06_EN );

			SPL07(	FeedBack_Contatore:=SPLIT07_ST ,SSPLIT_EN=> SPLIT07_EN );
			SPL08(	FeedBack_Contatore:=SPLIT08_ST ,SSPLIT_EN=> SPLIT08_EN );
			SPL09(	FeedBack_Contatore:=SPLIT09_ST ,SSPLIT_EN=> SPLIT09_EN );

			SPL10(	FeedBack_Contatore:=SPLIT10_ST ,SSPLIT_EN=> SPLIT10_EN );
			SPL11(	FeedBack_Contatore:=SPLIT11_ST ,SSPLIT_EN=> SPLIT11_EN );



END_IF

(*==============================*)
(*== System cycle operations ===*)
(*==============================*)
(* Execute TCP processes *)
Logger_Proc();
Remote_Proc();
(* Update user led *)
USRLED_Update();
(* Execute Cron Editor commands *)
CronEd();


(* Environment temperature *)
IF NOT TPV01.ERR THEN T_AMB := T_S01;
ELSE T_AMB := Plant_DefaultTAmb;
END_IF
END_PROGRAM
ACTION Main_Stm:
CASE Sys.Status OF

	S_STARTUP:
		Sys.Status:=S_INIT_RTC;

	S_INIT_RTC:
		(* Check RTC and update from network *)
		RTC_Update();
		(* Check time *)
		IF Sys.Time_Year>2000 THEN
			Sys.Status:=S_INIT_VAR;
		END_IF

	S_INIT_VAR:
		LogEv(EL_Wrn,EO_SYS,0,1,CONCAT('System_startup_v',WORD_TO_STRING(Plant_SW_VER)));
		Sys.Status:=S_RUNNING;

	S_RUNNING:
		Timer1(IN:=NOT Timer1.Q,PT:=T#50ms);
		IF Timer1.Q THEN
			(* Update meters *)
			CTL01 ( CTL_ST:=CTL01_ST, COUNT:=CTL01_Count );
			(* Update system checks *)
			SYS_Proc();
		END_IF

		Timer2(IN:=NOT Timer2.Q,PT:=T#500ms);
		IF Timer2.Q THEN
			(* Read current date/time *)
			RTC_Update();
			(* Execute plant operations *)
			TPV01	 ( IN:=T_S01 );
			TPV02	 ( IN:=T_S02 );
			TPV03	 ( IN:=T_S03 );
			TPV04	 ( IN:=T_S04 );
			TPV05	 ( IN:=T_S05 );
			TPV06	 ( IN:=T_S06 );
			TPV07	 ( IN:=T_S07 );
			TPV08	 ( IN:=T_S08 );
			TPV09	 ( IN:=T_S09 );
			TPV10	 ( IN:=T_S10 );
			TPV11	 ( IN:=T_S11 );

			TAMB  ( IN1:=TPV01, IN2:=TPV01 );


			(* Crono Termnostati  *)
			THER01(Temperature:=TPV10.AVG);
			SPL10.Split_RUN:=SEL(TPV10.ERR,THER01.Run,THER01.RunCrono); (* Piano Palestrina Alto *)
			SPL11.Split_RUN:=SEL(TPV10.ERR,THER01.Run,THER01.RunCrono); (* Piano Palestrina Basso *)

			(* per questi SPLIT è previsto la partenza in alternata quindi scambio l'isteresi locale tutte le volte che il conto spegne *)

			TrigR_THER01(clk:=THER01.Run);
			IF TrigR_THER01.Q THEN
				VarApp:=SPL10.TempIsteresiLocale;
				SPL10.TempIsteresiLocale:=SPL11.TempIsteresiLocale;
				SPL11.TempIsteresiLocale:=VarApp;
			END_IF



			(* Sicurezze e comandi *)
		 	SPL10(TemperaturaRiferimento:=THER01.Temperature,TemperaturaSet:=THER01.SetPoint,LimiteIsteresi:=THER01.Histeresys,TemperaturaOK:=TPV05.AVG>SPL10.SogliaTemperaturaMandata);
	 		SPL11(TemperaturaRiferimento:=THER01.Temperature,TemperaturaSet:=THER01.SetPoint,LimiteIsteresi:=THER01.Histeresys,TemperaturaOK:=TPV05.AVG>SPL11.SogliaTemperaturaMandata);


			(* Crono Termnostati  *)
			THER02(Temperature:=TPV08.AVG);
			SPL04.Split_RUN:=SEL(TPV08.ERR,THER02.Run,THER02.RunCrono); (* Palestra Lato SX Alto *)
			SPL05.Split_RUN:=SEL(TPV08.ERR,THER02.Run,THER02.RunCrono); (* Palestra Lato SX Centro *)
			SPL06.Split_RUN:=SEL(TPV08.ERR,THER02.Run,THER02.RunCrono); (* Palestra Lato SX Basso *)

			(* Sicurezze e comandi *)
		 	SPL04(TemperaturaRiferimento:=THER02.Temperature,TemperaturaSet:=THER02.SetPoint,LimiteIsteresi:=THER02.Histeresys,TemperaturaOK:=TPV05.AVG>SPL04.SogliaTemperaturaMandata);
	 		SPL05(TemperaturaRiferimento:=THER02.Temperature,TemperaturaSet:=THER02.SetPoint,LimiteIsteresi:=THER02.Histeresys,TemperaturaOK:=TPV05.AVG>SPL05.SogliaTemperaturaMandata);
	 		SPL06(TemperaturaRiferimento:=THER02.Temperature,TemperaturaSet:=THER02.SetPoint,LimiteIsteresi:=THER02.Histeresys,TemperaturaOK:=TPV05.AVG>SPL06.SogliaTemperaturaMandata);

			(* Crono Termnostati  *)
			THER03(Temperature:=TPV09.AVG);
			SPL07.Split_RUN:=SEL(TPV09.ERR,THER03.Run,THER03.RunCrono); (* Palestra Lato DX Alto *)
			SPL08.Split_RUN:=SEL(TPV09.ERR,THER03.Run,THER03.RunCrono); (* Palestra Lato DX Centro *)
			SPL09.Split_RUN:=SEL(TPV09.ERR,THER03.Run,THER03.RunCrono); (* Palestra Lato DX Basso *)

			(* Sicurezze e comandi *)
		 	SPL07(TemperaturaRiferimento:=THER03.Temperature,TemperaturaSet:=THER03.SetPoint,LimiteIsteresi:=THER03.Histeresys,TemperaturaOK:=TPV05.AVG>SPL07.SogliaTemperaturaMandata);
	 		SPL08(TemperaturaRiferimento:=THER03.Temperature,TemperaturaSet:=THER03.SetPoint,LimiteIsteresi:=THER03.Histeresys,TemperaturaOK:=TPV05.AVG>SPL08.SogliaTemperaturaMandata);
	 		SPL09(TemperaturaRiferimento:=THER03.Temperature,TemperaturaSet:=THER03.SetPoint,LimiteIsteresi:=THER03.Histeresys,TemperaturaOK:=TPV05.AVG>SPL09.SogliaTemperaturaMandata);

			(* Crono Termnostati  *)
			THER04(Temperature:=TPV11.AVG);
			SPL01.Split_RUN:=SEL(TPV11.ERR,THER04.Run,THER04.RunCrono); (* Gradinata Lato SX *)
			SPL02.Split_RUN:=SEL(TPV11.ERR,THER04.Run,THER04.RunCrono); (* Gradinata Lato Centro *)
			SPL03.Split_RUN:=SEL(TPV11.ERR,THER04.Run,THER04.RunCrono); (* Gradinata Lato DX *)

			(* Sicurezze e comandi *)
		 	SPL01(TemperaturaRiferimento:=THER04.Temperature,TemperaturaSet:=THER04.SetPoint,LimiteIsteresi:=THER04.Histeresys,TemperaturaOK:=TPV05.AVG>SPL01.SogliaTemperaturaMandata);
	 		SPL02(TemperaturaRiferimento:=THER04.Temperature,TemperaturaSet:=THER04.SetPoint,LimiteIsteresi:=THER04.Histeresys,TemperaturaOK:=TPV05.AVG>SPL02.SogliaTemperaturaMandata);
	 		SPL03(TemperaturaRiferimento:=THER04.Temperature,TemperaturaSet:=THER04.SetPoint,LimiteIsteresi:=THER04.Histeresys,TemperaturaOK:=TPV05.AVG>SPL03.SogliaTemperaturaMandata);






		(* Ciroclatore  Assevito agli SPLIT *)
			(* comndato dai vari cronotermostati *)
			CIRD04.OnOff:=THER01.Run OR THER02.Run
							OR THER03.Run OR THER04.Run;
	(*		(* comandato dai vari crono *)
			CIRD04.OnOff:=THER01.RunCrono OR THER02.RunCrono
							OR THER03.RunCrono OR THER04.RunCrono; *)

			(* Crono  *)
			THER05();
			CIRD05.OnOff:=THER05.RunCrono; (* Servizi *)

			(* Crono Termnostati  *)
			THER06(Temperature:=TPV04.AVG);
			CIRD02.OnOff:=SEL(TPV06.ERR,THER06.Run,THER06.RunCrono); (* Bollitore *)

			(* Crono  *)
			THER07();
			CIRD03.OnOff:=THER07.RunCrono; (* Servizi *)

			(*  l'offset Boost viene fatto direttamente sulle cliamtiche delle VRD perchè nonesiste la curva cliamtica della caldaia *)
			VRD01(RUN:=TRUE,CLIM:=VRD01_Clima,OffsetBoost:=THER250.SetPoint, TEMP:=TPV07.AVG, STATUS:=VRD01_ST, OUT=>VRD01_CTRL);
			VRD02(RUN:=CIRD04.Run, CLIM:=VRD02_Clima,OffsetBoost:=THER250.SetPoint, TEMP:=TPV05.AVG, STATUS:=VRD02_ST, OUT=>VRD02_CTRL);
			VRD03(RUN:=CIRD05.Run, CLIM:=VRD03_Clima,OffsetBoost:=THER250.SetPoint, TEMP:=TPV06.AVG, STATUS:=VRD03_ST, OUT=>VRD03_CTRL);


			THER250();



			(* Ciroclatore Primario Caldaia *)
			CIRD01.OnOff:=( CIRD02.Ctrl_Run OR CIRD04.Ctrl_Run OR CIRD05.Ctrl_Run ) AND SYS.AlarmStop=FALSE;

			(* Caldaia in RUN *)

			CAL01.Run := CIRD01.OnOff;


			(* Set Point Caldaia *)
			CAL01.SetPointManuale:=CAL01.Curve_Temp - OffsetSetPointManuale + THER250.SetPoint;  	(* Temperatrura del Boost *)

			CAL01.SetPointManuale:=MAX(CAL01.SetPointManuale,SEL(CIRD02.OnOff,0,THER06.SetPoint + OffsetSetPointManuale));
			CAL01.SetPointManuale:=MAX(CAL01.SetPointManuale,SEL(VRD01.RUN,0,VRD01.Ctrl_SetPoint));
			CAL01.SetPointManuale:=MAX(CAL01.SetPointManuale,SEL(VRD02.RUN,0,VRD02.Ctrl_SetPoint));
			CAL01.SetPointManuale:=MAX(CAL01.SetPointManuale,SEL(VRD03.RUN,0,VRD03.Ctrl_SetPoint));

			CAL01(CLIM:=CAL01_Clima,AbilitaSetPointManuale:=TRUE);


			Lamp( Allarme:=	(CAL01.Status_Log=2) OR
  						  	CIRD01.Status_Log=2 OR
  						  	CIRD02.Status_Log=2 OR
  						  	CIRD03.Status_Log=2 OR
 						  	CIRD04.Status_Log=2 OR
						  	CIRD05.Status_Log=2 OR
							TPV01.Status_Log=2 OR
							TPV02.Status_Log=2 OR
							TPV03.Status_Log=2 OR
							TPV04.Status_Log=2 OR
							TPV05.Status_Log=2 OR
							TPV06.Status_Log=2 OR
							TPV07.Status_Log=2 OR
							TPV08.Status_Log=2 OR
							TPV09.Status_Log=2 OR
							TPV10.Status_Log=2 OR
							TPV11.Status_Log=2 OR
							THER01.Status_Log=2 OR
							THER02.Status_Log=2 OR
							THER03.Status_Log=2 OR
							THER04.Status_Log=2 OR
							THER250.Status_Log=2 OR
							VRD01.Status_Log=2 OR
							VRD02.Status_Log=2 OR
							VRD03.Status_Log=2 OR
							SPL01.Status_Log=2 OR
							SPL01.Status_Log=2 OR
							SPL02.Status_Log=2 OR
							SPL03.Status_Log=2 OR
							SPL04.Status_Log=2 OR
							SPL05.Status_Log=2 OR
							SPL06.Status_Log=2 OR
							SPL07.Status_Log=2 OR
							SPL08.Status_Log=2 OR
							SPL09.Status_Log=2 OR
							SPL10.Status_Log=2 OR
							SPL11.Status_Log=2
							,
							Warning:=	(CAL01.Status_Log=1) OR
  						  	CIRD01.Status_Log=1 OR
  						  	CIRD02.Status_Log=1 OR
  						  	CIRD03.Status_Log=1 OR
 						  	CIRD04.Status_Log=1 OR
						  	CIRD05.Status_Log=1 OR
							TPV01.Status_Log=1 OR
							TPV02.Status_Log=1 OR
							TPV03.Status_Log=1 OR
							TPV04.Status_Log=1 OR
							TPV05.Status_Log=1 OR
							TPV06.Status_Log=1 OR
							TPV07.Status_Log=1 OR
							TPV08.Status_Log=1 OR
							TPV09.Status_Log=1 OR
							TPV10.Status_Log=1 OR
							TPV11.Status_Log=1 OR
							THER01.Status_Log=1 OR
							THER02.Status_Log=1 OR
							THER03.Status_Log=1 OR
							THER04.Status_Log=1 OR
							THER250.Status_Log=1 OR
							VRD01.Status_Log=1 OR
							VRD02.Status_Log=1 OR
							VRD03.Status_Log=1 OR
							SPL01.Status_Log=1 OR
							SPL01.Status_Log=1 OR
							SPL02.Status_Log=1 OR
							SPL03.Status_Log=1 OR
							SPL04.Status_Log=1 OR
							SPL05.Status_Log=1 OR
							SPL06.Status_Log=1 OR
							SPL07.Status_Log=1 OR
							SPL08.Status_Log=1 OR
							SPL09.Status_Log=1 OR
							SPL10.Status_Log=1 OR
							SPL11.Status_Log=1
							,
							AllarmeLampada=>LAMP_AL
							);



		END_IF

		Timer3(IN:=NOT Timer3.Q,PT:=T#5m);
		IF Timer3.Q OR HMI_AggiornaLog THEN
			(* Trig logger *)
			LogTrig();
			(* Execute temporary CSV logger *)
			CSV_Log();
		END_IF

	S_SHUTDOWN:
		(* Stop caldaia *)
		(* Stop deviatori *)
		(* Aspetta 5 min prima di spegnere eventuali circolatori *)
		Sys.Status:=S_STARTUP;

	S_HALT:
		(* Aspetta uscita manuale *)
		Sys.Status:=S_STARTUP;


ELSE
	Sys.Status:=S_STARTUP;
END_CASE;
END_ACTION
ACTION NodoWAGO:
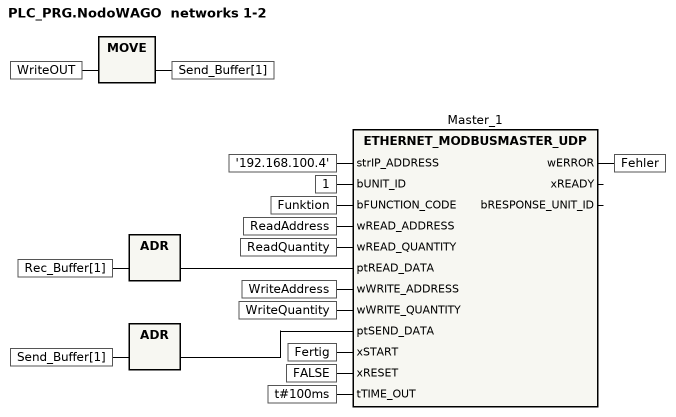
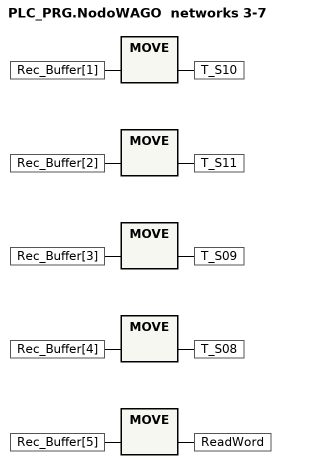
_FBD_ (* Function Block Diagram *)
NETWORK 1
	MOVE(WriteOUT) => Send_Buffer[1]
NETWORK 2
	Master_1:ETHERNET_MODBUSMASTER_UDP(strIP_ADDRESS: '192.168.100.4', bUNIT_ID: 1, bFUNCTION_CODE: Funktion, wREAD_ADDRESS: ReadAddress, wREAD_QUANTITY: ReadQuantity, ptREAD_DATA: ADR(Rec_Buffer[1]), wWRITE_ADDRESS: WriteAddress, wWRITE_QUANTITY: WriteQuantity, ptSEND_DATA: ADR(Send_Buffer[1]), xSTART: Fertig, xRESET: FALSE, tTIME_OUT: t#100ms) => Fehler
NETWORK 3
	MOVE(Rec_Buffer[1]) => T_S10
NETWORK 4
	MOVE(Rec_Buffer[2]) => T_S11
NETWORK 5
	MOVE(Rec_Buffer[3]) => T_S09
NETWORK 6
	MOVE(Rec_Buffer[4]) => T_S08
NETWORK 7
	MOVE(Rec_Buffer[5]) => ReadWord
_END_FBD_
(* the same logic as Structured Text *)
(* Network 1 *)
Send_Buffer[1] := WriteOUT;
(* Network 2 *)
Master_1(strIP_ADDRESS := '192.168.100.4', bUNIT_ID := 1, bFUNCTION_CODE := Funktion, wREAD_ADDRESS := ReadAddress, wREAD_QUANTITY := ReadQuantity, ptREAD_DATA := ADR(Rec_Buffer[1]), wWRITE_ADDRESS := WriteAddress, wWRITE_QUANTITY := WriteQuantity, ptSEND_DATA := ADR(Send_Buffer[1]), xSTART := Fertig, xRESET := FALSE, tTIME_OUT := t#100ms);
Fehler := Master_1.wERROR;
(* Network 3 *)
T_S10 := Rec_Buffer[1];
(* Network 4 *)
T_S11 := Rec_Buffer[2];
(* Network 5 *)
T_S09 := Rec_Buffer[3];
(* Network 6 *)
T_S08 := Rec_Buffer[4];
(* Network 7 *)
ReadWord := Rec_Buffer[5];
END_ACTION

(* POU LON/Module_1/Module_1_PRG, FBD *)
PROGRAM Module_1_PRG
VAR
	(* Automatic added code, do not change! *)
	LonMaster : Module_1_LonMaster;
	SFPTnodeObject : Module_1_SFPTnodeObject;
	Virtualfunctionalblock : Module_1_Virtualfunctionalblock;

	InData_LON AT %IB0 : ARRAY[0..23] OF BYTE;
	OutData_LON AT %QB0 : ARRAY[0..23] OF BYTE;
	(***** End of automatic added code. *****)

	(* Add your code here. *)

END_VAR
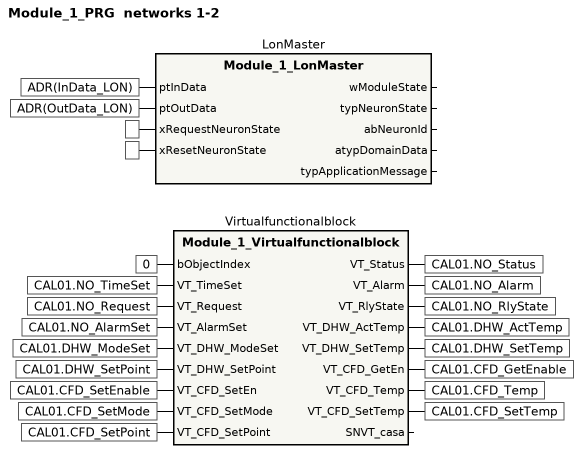
_FBD_ (* Function Block Diagram *)
NETWORK 1 (* Added by code generator *)
	LonMaster:Module_1_LonMaster(ptInData: ADR(InData_LON), ptOutData: ADR(OutData_LON), xRequestNeuronState: , xResetNeuronState: )
NETWORK 2
	Virtualfunctionalblock:Module_1_Virtualfunctionalblock(bObjectIndex: 0, VT_TimeSet: CAL01.NO_TimeSet, VT_Request: CAL01.NO_Request, VT_AlarmSet: CAL01.NO_AlarmSet, VT_DHW_ModeSet: CAL01.DHW_ModeSet, VT_DHW_SetPoint: CAL01.DHW_SetPoint, VT_CFD_SetEn: CAL01.CFD_SetEnable, VT_CFD_SetMode: CAL01.CFD_SetMode, VT_CFD_SetPoint: CAL01.CFD_SetPoint, VT_Alarm => CAL01.NO_Alarm, VT_RlyState => CAL01.NO_RlyState, VT_DHW_ActTemp => CAL01.DHW_ActTemp, VT_DHW_SetTemp => CAL01.DHW_SetTemp, VT_CFD_GetEn => CAL01.CFD_GetEnable, VT_CFD_Temp => CAL01.CFD_Temp, VT_CFD_SetTemp => CAL01.CFD_SetTemp) => CAL01.NO_Status
_END_FBD_
(* the same logic as Structured Text *)
(* Network 1: see the listing above *)
(* Network 2 *)
Virtualfunctionalblock(bObjectIndex := 0, VT_TimeSet := CAL01.NO_TimeSet, VT_Request := CAL01.NO_Request, VT_AlarmSet := CAL01.NO_AlarmSet, VT_DHW_ModeSet := CAL01.DHW_ModeSet, VT_DHW_SetPoint := CAL01.DHW_SetPoint, VT_CFD_SetEn := CAL01.CFD_SetEnable, VT_CFD_SetMode := CAL01.CFD_SetMode, VT_CFD_SetPoint := CAL01.CFD_SetPoint);
CAL01.NO_Alarm := Virtualfunctionalblock.VT_Alarm;
CAL01.NO_RlyState := Virtualfunctionalblock.VT_RlyState;
CAL01.DHW_ActTemp := Virtualfunctionalblock.VT_DHW_ActTemp;
CAL01.DHW_SetTemp := Virtualfunctionalblock.VT_DHW_SetTemp;
CAL01.CFD_GetEnable := Virtualfunctionalblock.VT_CFD_GetEn;
CAL01.CFD_Temp := Virtualfunctionalblock.VT_CFD_Temp;
CAL01.CFD_SetTemp := Virtualfunctionalblock.VT_CFD_SetTemp;
CAL01.NO_Status := Virtualfunctionalblock.VT_Status;
END_PROGRAM

(* POU LON/Module_1/Master/Module_1_LonMaster, ST *)
FUNCTION_BLOCK Module_1_LonMaster
(******************************************)
(* Automatic generated code, do not edit! *)
(******************************************)
VAR_INPUT
	ptInData  : POINTER TO BYTE;
	ptOutData : POINTER TO BYTE;
	xRequestNeuronState : BOOL;
	xResetNeuronState : BOOL;
END_VAR
VAR_OUTPUT
	wModuleState : WORD; (* bit coded wModuleState:
	15: communication to I/O-module interrupted (error)
	14 - 08: reserved
	07: ready for Neuron initialization
	06: Neuron active
	05: user interface active
	04: internal module communication interrupted (error)
	03: CP synchronization running
	02: Neuron is configured online
	01 - 00: reserved *)

	typNeuronState : NeuronState;
	abNeuronId : ARRAY[0..5] OF BYTE;
	atypDomainData : ARRAY[0..1] OF DomainData;
	typApplicationMessage : ApplicationMessageData;
END_VAR
VAR
	bInternalCode : BYTE;
	bNvIndex : BYTE;
	wCpIndex : WORD;
	lonCom : FbLonBasicCommunication;

	xInitIsStarted : BOOL := FALSE;

	TimeoutTimer : TON;
	timeOutTime : TIME := T#1000ms;
	xStateMachineIsChecked : BOOL;
	xTimerStart : BOOL;

	iDomainTable : INT;
	xSendRequestPending : BOOL;
	trigRequest : R_TRIG;
	trigReset : R_TRIG;

	abMbxRxPrio0Buf: ARRAY [0..309] OF BYTE;
	abMbxRxPrio1Buf: ARRAY [0..517] OF BYTE;
	aMbxRxBufSize: ARRAY [0..1] OF UINT := 310, 518;
	aMbxRxBufList: ARRAY [0..1] OF POINTER TO BYTE;
	afbMbxRxFb: ARRAY [0..1] OF MBX2_RX_DEFRAG;
	astMbxRxCtx: ARRAY [0..1] OF stMbx2DefragContext;

	abMbxTxPrio0Buf: ARRAY [0..309] OF BYTE;
	abMbxTxPrio1Buf: ARRAY [0..517] OF BYTE;
	aMbxTxBufSize: ARRAY [0..1] OF UINT := 310, 518;
	aMbxTxBufList: ARRAY [0..1] OF POINTER TO BYTE;
	afbMbxTxFb: ARRAY [0..1] OF MBX2_TX_FRAG;

	astMbxTrackContext: ARRAY [0..0] OF stMbx2TrackContext;
END_VAR
VAR CONSTANT
END_VAR
aMbxRxBufList[0] := ADR(abMbxRxPrio0Buf[0]);
aMbxRxBufList[1] := ADR(abMbxRxPrio1Buf[0]);

aMbxTxBufList[0] := ADR(abMbxTxPrio0Buf[0]);
aMbxTxBufList[1] := ADR(abMbxTxPrio1Buf[0]);

mbxModule_1.Ressources.pDefragBufList := ADR(aMbxRxBufList);
mbxModule_1.Ressources.pDefragBufSizeList := ADR(aMbxRxBufSize);
mbxModule_1.Ressources.pDefragCtxPtrList := ADR(astMbxRxCtx);
mbxModule_1.Ressources.pDefragFbList := ADR(afbMbxRxFb);
mbxModule_1.Ressources.pFragBufList := ADR(aMbxTxBufList);
mbxModule_1.Ressources.pFragBufSizeList := ADR(aMbxTxBufSize);
mbxModule_1.Ressources.pFragFbList := ADR(afbMbxTxFb);

mbxModule_1.Ressources.unMaxAvailableRxPrioIndex := 1;
mbxModule_1.Ressources.unMaxAvailableTxPrioIndex := 1;

mbxModule_1.Ressources.pTrackStList := ADR(astMbxTrackContext);
mbxModule_1.Ressources.unMaxAvailableTrackIndex := 0;

mbxModule_1.Ressources.pabRxWin := ptInData + 1;
mbxModule_1.Ressources.pabTxWin := ptOutData + 1;
mbxModule_1.Ressources.bTxWinSize := 23;
mbxModule_1.Ressources.bRxWinSize := 23;

IF (mbxModule_1.bStatus.2 = TRUE) OR (mbxModule_1.bStatus.1 = TRUE) THEN
	mbxModule_1.MBX_RESET();
	xInitRunning_Module_1 := TRUE;
	xInitIsStarted := FALSE;
END_IF
mbxModule_1.MBX_CYCLE();

IF (mbxModule_1.bStatus.0 <> TRUE) THEN 
	wModuleState := 16#8000;
	RETURN;
ELSE
	wModuleState.15 := FALSE;
END_IF

xStateMachineIsChecked := FALSE;
IF xInitRunning_Module_1 = TRUE THEN
	IF xInitIsStarted = FALSE THEN
		SetParameter();
		lonCom.eInitState := INIT_SND_SGNTR_REQ;
		lonCom.CheckInitState();
		xInitIsStarted := TRUE;
		xStateMachineIsChecked := TRUE;
	END_IF
END_IF

typApplicationMessage.xMsgRcvd := FALSE;
typApplicationMessage.xRspRcvd := FALSE;
ResetNviUpdate();
WHILE (mbxModule_1.xRxPending) DO
	unLastLen_mbxModule_1 := mbxModule_1.unRxLen;
	mbxModule_1.pbRxData := ADR(InDataTelegram_Module_1);
	mbxModule_1.MBX_RETRIEVE();
	IF (mbxModule_1.nError <> MBX_OK) THEN EXIT; END_IF;
	bInternalCode := InDataTelegram_Module_1[0];

	IF (xInitRunning_Module_1 = TRUE) AND (lonCom.eInitState <> INIT_TRANSFER_CFG) THEN
		IF (FuCheckForValidInitCode(bInternalCode)) THEN
			SetParameter();
			lonCom.unLastLen := unLastLen_mbxModule_1;
			lonCom.CheckInitState();
			xInitRunning_Module_1 := NOT lonCom.xInitDone;
			xStateMachineIsChecked := TRUE;
		END_IF
	END_IF

	IF (bInternalCode = M2C_NVI_UPDT_OCCD) OR (bInternalCode = M2C_NV_VALUE_RSP) OR (bInternalCode = M2C_NVI_UPDT_TOUT) THEN
		bNvIndex := InDataTelegram_Module_1[1];
		CASE bNvIndex OF
			0, 2, 4: Module_1_PRG.SFPTnodeObject.DataReceived();
			13..21: Module_1_PRG.Virtualfunctionalblock.DataReceived();

		END_CASE;
	ELSIF (bInternalCode = M2C_CP_VALUE_RSP) THEN
		wCpIndex := InDataTelegram_Module_1[1] OR (InDataTelegram_Module_1[2] * 256);
		CASE wCpIndex OF

		END_CASE;
	ELSIF (bInternalCode = M2C_LON_MSG_RCVD) OR (bInternalCode = M2C_LON_RSP_RCVD) THEN
		ApplMsgReceived();
	ELSIF (bInternalCode = M2C_STATUS_RSP) THEN
		wModuleState := (wModuleState AND 16#FF00) + InDataTelegram_Module_1[1];
	ELSIF (bInternalCode = M2C_NEURON_ID) THEN
		FuMemCopy(ADR(InDataTelegram_Module_1[1]), ADR(abNeuronId), 6);
	ELSIF (bInternalCode = M2C_DOMAIN_DATA) THEN
		DomainDataRcvd();
	ELSIF (bInternalCode = M2C_MICRO_SERVER_STATUS_RSP) THEN
		NeuronStateRcvd();
	END_IF
END_WHILE

IF (xInitRunning_Module_1 = TRUE) AND ((lonCom.xCallStateMachine = TRUE) OR (TimeoutTimer.Q = TRUE)) AND (NOT xStateMachineIsChecked) THEN
	SetParameter();
	lonCom.xTimeOut := TimeoutTimer.Q;
	lonCom.CheckInitState();
END_IF
TimeoutTimer(IN:=lonCom.xTimerStart, PT:=timeOutTime);

trigRequest(CLK := xRequestNeuronState);
trigReset(CLK := xResetNeuronState);
IF (trigRequest.Q OR trigReset.Q) THEN
	RequestNeuronState();
END_IF
END_FUNCTION_BLOCK
ACTION ApplMsgReceived:
IF (InDataTelegram_Module_1[0] = M2C_LON_MSG_RCVD) THEN
	typApplicationMessage.typService := InDataTelegram_Module_1[1] AND 16#30;
	typApplicationMessage.bSourceSubnetId := InDataTelegram_Module_1[2];
	typApplicationMessage.bSourceNodeId := InDataTelegram_Module_1[3];
	typApplicationMessage.bCorrelator := InDataTelegram_Module_1[4];
	typApplicationMessage.bCode :=  InDataTelegram_Module_1[5];
	typApplicationMessage.bDataLength := UINT_TO_BYTE(unLastLen_mbxModule_1 - 6);
	IF typApplicationMessage.bDataLength > 48 THEN typApplicationMessage.bDataLength := 48; END_IF;
	FuMemSet(ADR(typApplicationMessage.abData), 0, SIZEOF(typApplicationMessage.abData));
	IF typApplicationMessage.bDataLength > 0 THEN
		FuMemCopy(ADR(InDataTelegram_Module_1[6]), ADR(typApplicationMessage.abData), typApplicationMessage.bDataLength);
	END_IF
	typApplicationMessage.xMsgRcvd := TRUE;
ELSE
	typApplicationMessage.typService := LON_RESPONSE;
	typApplicationMessage.bSourceSubnetId := InDataTelegram_Module_1[1];
	typApplicationMessage.bSourceNodeId := InDataTelegram_Module_1[2];
	typApplicationMessage.bCorrelator := 0;
	typApplicationMessage.bCode :=  InDataTelegram_Module_1[3];
	typApplicationMessage.bDataLength := UINT_TO_BYTE(unLastLen_mbxModule_1 - 4);
	IF typApplicationMessage.bDataLength > 48 THEN typApplicationMessage.bDataLength := 48; END_IF;
	FuMemSet(ADR(typApplicationMessage.abData), 0, SIZEOF(typApplicationMessage.abData));
	IF typApplicationMessage.bDataLength > 0 THEN
		FuMemCopy(ADR(InDataTelegram_Module_1[4]), ADR(typApplicationMessage.abData), typApplicationMessage.bDataLength);
	END_IF
	typApplicationMessage.xRspRcvd := TRUE;
END_IF
END_ACTION
ACTION DomainDataRcvd:
IF (unLastLen_mbxModule_1 = 17) THEN
	iDomainTable := InDataTelegram_Module_1[1];
	IF (iDomainTable < 0) OR (iDomainTable > 1) THEN RETURN; END_IF
	FuMemCopy(ADR(InDataTelegram_Module_1[2]), ADR(atypDomainData[iDomainTable].abDomainId), 6);
	atypDomainData[iDomainTable].bSubnet := InDataTelegram_Module_1[8];
	atypDomainData[iDomainTable].xIsNonClone := InDataTelegram_Module_1[9].7;
	atypDomainData[iDomainTable].bNodeId := InDataTelegram_Module_1[9] AND 16#7F;
	atypDomainData[iDomainTable].xIsInvalid := InDataTelegram_Module_1[10].7;
	atypDomainData[iDomainTable].bDomainIdLength := InDataTelegram_Module_1[10] AND 16#7F;
	FuMemCopy(ADR(InDataTelegram_Module_1[11]), ADR(atypDomainData[iDomainTable].abAuthenticationKey), 6);
END_IF
END_ACTION
ACTION NeuronStateRcvd:
IF (unLastLen_mbxModule_1 = 16) THEN
	typNeuronState.wCrcError := InDataTelegram_Module_1[1] + InDataTelegram_Module_1[2] * 256;
	typNeuronState.wTransactionTimeouts := InDataTelegram_Module_1[3] + InDataTelegram_Module_1[4] * 256;
	typNeuronState.wReceiveTransactionBuffersFull := InDataTelegram_Module_1[5] + InDataTelegram_Module_1[6] * 256;
	typNeuronState.wLostMessages := InDataTelegram_Module_1[7] + InDataTelegram_Module_1[8] * 256;
	typNeuronState.wMissedMessages := InDataTelegram_Module_1[9] + InDataTelegram_Module_1[10] * 256;
	typNeuronState.bResetCause := InDataTelegram_Module_1[11];
	typNeuronState.bNodeState := InDataTelegram_Module_1[12];
	typNeuronState.bFirmwareVersion := InDataTelegram_Module_1[13];
	typNeuronState.bLastErrorLogged := InDataTelegram_Module_1[14];
	typNeuronState.bModelNumber := InDataTelegram_Module_1[15];
END_IF
END_ACTION
ACTION RequestNeuronState:
OutDataTelegram_Module_1[0] := C2M_MICRO_SERVER_STATUS_QRY;
OutDataTelegram_Module_1[1] := BOOL_TO_BYTE(trigReset.Q);

mbxModule_1.bTxPrio := 1;
mbxModule_1.bTxProtID := 0;
mbxModule_1.pbTxData := ADR(OutDataTelegram_Module_1);
mbxModule_1.unTxLen := 2;
mbxModule_1.MBX_SEND();

IF (mbxModule_1.nError <> MBX_OK) THEN
	RETURN;
END_IF
END_ACTION
ACTION ResetNviUpdate:
Module_1_PRG.SFPTnodeObject.ResetNviUpdate();
Module_1_PRG.Virtualfunctionalblock.ResetNviUpdate();
END_ACTION
ACTION SetParameter:
lonCom.pMbx 			:= ADR(mbxModule_1);
lonCom.pInData 			:= ADR(InDataTelegram_Module_1);
lonCom.pOutData 		:= ADR(OutDataTelegram_Module_1);
lonCom.pTimer			:= ADR(TimeoutTimer);

lonCom.pActualSignature	:= ADR(abSignature_Module_1);
lonCom.pConfigBlock := ADR(abInterface_Module_1);
lonCom.wConfigSize 		:= wConfigSize_Module_1;
END_ACTION

(* POU LON/Module_1/NV_Interface/Module_1_SFPTnodeObject, ST *)
FUNCTION_BLOCK Module_1_SFPTnodeObject
(******************************************)
(* Automatic generated code, do not edit! *)
(******************************************)
VAR_INPUT
	bObjectIndex : BYTE := 0;
	nvoStatus : typSnvtObjStatus;
	nvoFileStat : typSnvtFileStatus;

END_VAR
VAR_OUTPUT
	nviRequest : typSnvtObjRequest;
	nviFileReq : typSnvtFileReq;
	nviFilePos : typSnvtFilePos;

END_VAR
VAR
	xSetOnce : BOOL := TRUE;
	xDataInUpdated : BOOL := FALSE;
	nvoStatusLast: typSnvtObjStatus;
	nvoFileStatLast: typSnvtFileStatus;

	cmd : BYTE;
	z : INT;
	bNvRelativeIdx : BYTE;
	bNvAbsoluteIdx : BYTE;
	wCpRelativeIdx : WORD;
	wCpAbsoluteIdx : WORD;
END_VAR
VAR CONSTANT
	bNvStartIndex : BYTE := 0;
	wCpStartIndex : WORD := 65535;
	bLmoCount : BYTE := 1;
END_VAR
IF (xInitRunning_Module_1 = TRUE) AND (xSetOnce = TRUE) THEN
	xSetOnce := FALSE;
	CachePointers();
	SetUpdateFlags();
END_IF

CheckUpdateFlags();
IF (xInitRunning_Module_1 = FALSE) AND (xDataInUpdated = FALSE) THEN
	IF (mbxModule_1.bStatus.0) THEN
		SendValueRequest();
	END_IF
END_IF

IF (xInitRunning_Module_1 = FALSE) AND (mbxModule_1.bStatus.0) THEN
	xSetOnce := TRUE;
	xDataInUpdated := FALSE;
	IF ((NOT FuMemCompare(ADR(nvoStatusLast), ADR(nvoStatus), ADR(nvoStatus.bStatusInformation) - ADR(nvoStatus))) OR (nvoStatus.bStatusInformation.7 = TRUE) OR (nvoStatusLast.bInternalUseOnly.1 = TRUE)) THEN
		FuSnvtObjStatusToRaw(ADR(nvoStatus), ADR(OutDataTelegram_Module_1[2]));

		bNvAbsoluteIdx := bNvStartIndex + bObjectIndex + (1 * bLmoCount);

		IF (FuDoNvoUpdate_Module_1(ADR(nvoStatus), ADR(nvoStatusLast), ADR(nvoStatus.bInternalUseOnly), ADR(nvoStatusLast.bInternalUseOnly), ADR(nvoStatus.bStatusInformation), bNvAbsoluteIdx, 6, SIZEOF(nvoStatus)) = FALSE) THEN
			RETURN;
		END_IF
	END_IF
	IF ((NOT FuMemCompare(ADR(nvoFileStatLast), ADR(nvoFileStat), ADR(nvoFileStat.bStatusInformation) - ADR(nvoFileStat))) OR (nvoFileStat.bStatusInformation.7 = TRUE) OR (nvoFileStatLast.bInternalUseOnly.1 = TRUE)) THEN
		FuSnvtFileStatusToRaw(ADR(nvoFileStat), ADR(OutDataTelegram_Module_1[2]));

		bNvAbsoluteIdx := bNvStartIndex + bObjectIndex + (3 * bLmoCount);

		IF (FuDoNvoUpdate_Module_1(ADR(nvoFileStat), ADR(nvoFileStatLast), ADR(nvoFileStat.bInternalUseOnly), ADR(nvoFileStatLast.bInternalUseOnly), ADR(nvoFileStat.bStatusInformation), bNvAbsoluteIdx, 27, SIZEOF(nvoFileStat)) = FALSE) THEN
			RETURN;
		END_IF
	END_IF

END_IF
END_FUNCTION_BLOCK
ACTION CachePointers:
;
END_ACTION
ACTION CheckUpdateFlags:
xDataInUpdated := (NOT nviRequest.bInternalUseOnly.0) AND (NOT nviFileReq.bInternalUseOnly.0) AND (NOT nviFilePos.bInternalUseOnly.0) AND TRUE;
END_ACTION
ACTION DataReceived:
cmd := InDataTelegram_Module_1[0];
IF (cmd = M2C_NVI_UPDT_OCCD) OR (cmd = M2C_NV_VALUE_RSP) OR (cmd = M2C_NVI_UPDT_TOUT) THEN
	bNvRelativeIdx := (InDataTelegram_Module_1[1] - bNvStartIndex - bObjectIndex) / bLmoCount;
	CASE bNvRelativeIdx OF
	0:
		IF (cmd = M2C_NVI_UPDT_OCCD) OR (cmd = M2C_NV_VALUE_RSP) THEN
			IF (unLastLen_mbxModule_1 = (2 + 3)) THEN
				FuRawToSnvtObjRequest(ADR(InDataTelegram_Module_1[2]), ADR(nviRequest));
				nviRequest.bInternalUseOnly.0 := FALSE;
				nviRequest.bStatusInformation := FuInkrementNviStatus(nviRequest.bStatusInformation);
			ELSIF (unLastLen_mbxModule_1 = 2) THEN
				nviRequest.bStatusInformation := FuInkrementNviStatus(nviRequest.bStatusInformation);
			END_IF
		ELSIF (cmd = M2C_NVI_UPDT_TOUT) THEN
			IF (unLastLen_mbxModule_1 = 3) THEN
				nviRequest.bStatusInformation.4 := BYTE_TO_BOOL(InDataTelegram_Module_1[2]);
			END_IF
		END_IF
	2:
		IF (cmd = M2C_NVI_UPDT_OCCD) OR (cmd = M2C_NV_VALUE_RSP) THEN
			IF (unLastLen_mbxModule_1 = (2 + 12)) THEN
				FuRawToSnvtFileReq(ADR(InDataTelegram_Module_1[2]), ADR(nviFileReq));
				nviFileReq.bInternalUseOnly.0 := FALSE;
				nviFileReq.bStatusInformation := FuInkrementNviStatus(nviFileReq.bStatusInformation);
			ELSIF (unLastLen_mbxModule_1 = 2) THEN
				nviFileReq.bStatusInformation := FuInkrementNviStatus(nviFileReq.bStatusInformation);
			END_IF
		ELSIF (cmd = M2C_NVI_UPDT_TOUT) THEN
			IF (unLastLen_mbxModule_1 = 3) THEN
				nviFileReq.bStatusInformation.4 := BYTE_TO_BOOL(InDataTelegram_Module_1[2]);
			END_IF
		END_IF
	4:
		IF (cmd = M2C_NVI_UPDT_OCCD) OR (cmd = M2C_NV_VALUE_RSP) THEN
			IF (unLastLen_mbxModule_1 = (2 + 6)) THEN
				FuRawToSnvtFilePos(ADR(InDataTelegram_Module_1[2]), ADR(nviFilePos));
				nviFilePos.bInternalUseOnly.0 := FALSE;
				nviFilePos.bStatusInformation := FuInkrementNviStatus(nviFilePos.bStatusInformation);
			ELSIF (unLastLen_mbxModule_1 = 2) THEN
				nviFilePos.bStatusInformation := FuInkrementNviStatus(nviFilePos.bStatusInformation);
			END_IF
		ELSIF (cmd = M2C_NVI_UPDT_TOUT) THEN
			IF (unLastLen_mbxModule_1 = 3) THEN
				nviFilePos.bStatusInformation.4 := BYTE_TO_BOOL(InDataTelegram_Module_1[2]);
			END_IF
		END_IF

	END_CASE
ELSIF (cmd = M2C_CP_VALUE_RSP) THEN
	wCpRelativeIdx := ((InDataTelegram_Module_1[1] + InDataTelegram_Module_1[2] * 256) - wCpStartIndex - bObjectIndex) / bLmoCount;
	CASE wCpRelativeIdx OF

	END_CASE
END_IF
END_ACTION
ACTION ResetNviUpdate:
nviRequest.bStatusInformation := nviRequest.bStatusInformation AND 16#F8;
nviFileReq.bStatusInformation := nviFileReq.bStatusInformation AND 16#F8;
nviFilePos.bStatusInformation := nviFilePos.bStatusInformation AND 16#F8;
;
END_ACTION
ACTION SendValueRequest:
IF (FuSendNviValueReq_Module_1(ADR(nviRequest.bInternalUseOnly), bNvStartIndex + bObjectIndex + (0 * bLmoCount)) = FALSE) THEN
	RETURN;
END_IF

IF (FuSendNviValueReq_Module_1(ADR(nviFileReq.bInternalUseOnly), bNvStartIndex + bObjectIndex + (2 * bLmoCount)) = FALSE) THEN
	RETURN;
END_IF

IF (FuSendNviValueReq_Module_1(ADR(nviFilePos.bInternalUseOnly), bNvStartIndex + bObjectIndex + (4 * bLmoCount)) = FALSE) THEN
	RETURN;
END_IF

;
END_ACTION
ACTION SetUpdateFlags:
nviRequest.bInternaluseOnly.0 := TRUE;
nvoStatusLast.bInternaluseOnly.1 := TRUE;
nvoStatusLast.bInternaluseOnly.7 := FALSE;
nviFileReq.bInternaluseOnly.0 := TRUE;
nvoFileStatLast.bInternaluseOnly.1 := TRUE;
nvoFileStatLast.bInternaluseOnly.7 := FALSE;
nviFilePos.bInternaluseOnly.0 := TRUE;
;
END_ACTION

(* POU LON/Shared/Internal/FuSnvtObjStatusToRaw, ST *)
FUNCTION FuSnvtObjStatusToRaw : BOOL
(******************************************)
(* Automatic generated code, do not edit! *)
(******************************************)
VAR_INPUT
	NvDataIn :  POINTER TO typSnvtObjStatus;
	DataOut : POINTER TO ARRAY[0..5] OF BYTE;
END_VAR
VAR
END_VAR
DataOut^[0] := WORD_TO_BYTE(SHR(NvDataIn^.wObjectId, 8));
DataOut^[1] := WORD_TO_BYTE(NvDataIn^.wObjectId);

DataOut^[2] := NvDataIn^.bBitfieldByteOffset2;

DataOut^[3] := NvDataIn^.bBitfieldByteOffset3;

DataOut^[4] := NvDataIn^.bBitfieldByteOffset4;

DataOut^[5] := NvDataIn^.bBitfieldByteOffset5;

FuSnvtObjStatusToRaw := TRUE;
END_FUNCTION

(* POU LON/Module_1/Internal/FuDoNvoUpdate_Module_1, ST *)
FUNCTION FuDoNvoUpdate_Module_1 : BOOL
(******************************************)
(* Automatic generated code, do not edit! *)
(******************************************)
VAR_INPUT
	ptNvo : POINTER TO BYTE;
	ptNvoLast : POINTER TO BYTE;
	ptNvoInternalUse : POINTER TO BYTE;
	ptNvoLastInternalUse : POINTER TO BYTE;
	ptNvoStatusInformation : POINTER TO BYTE;
	bNvoIndex : BYTE;
	uiNvoLength : UINT;
	uiNvoVariableLength : UINT;
END_VAR
IF (ptNvoLastInternalUse^.1 = TRUE) AND (ptNvoStatusInformation^.7 = FALSE) THEN
	OutDataTelegram_Module_1[0] := C2M_NV_VALUE;
ELSE
	OutDataTelegram_Module_1[0] := C2M_NVO_PROPAGATE;
END_IF
OutDataTelegram_Module_1[1] := bNvoIndex;

mbxModule_1.bTxPrio := BOOL_TO_BYTE(ptNvoLastInternalUse^.7);
mbxModule_1.bTxProtID := 0;
mbxModule_1.pbTxData := ADR(OutDataTelegram_Module_1);
mbxModule_1.unTxLen := 2 + uiNvoLength;
mbxModule_1.MBX_SEND();

IF (mbxModule_1.nError <> MBX_OK) THEN
	FuDoNvoUpdate_Module_1 := FALSE;
	RETURN;
END_IF

ptNvoLastInternalUse^.1 := FALSE;
ptNvoInternalUse^ := ptNvoLastInternalUse^;
FuMemCopy(ptNvo, ptNvoLast, uiNvoVariableLength);

FuDoNvoUpdate_Module_1 := TRUE;
END_FUNCTION

(* POU LON/Shared/Internal/FuSnvtFileStatusToRaw, ST *)
FUNCTION FuSnvtFileStatusToRaw : BOOL
(******************************************)
(* Automatic generated code, do not edit! *)
(******************************************)
VAR_INPUT
	NvDataIn :  POINTER TO typSnvtFileStatus;
	DataOut : POINTER TO ARRAY[0..26] OF BYTE;
END_VAR
VAR
END_VAR
DataOut^[0] := NvDataIn^.bStatus;

DataOut^[1] := WORD_TO_BYTE(SHR(NvDataIn^.wNumberOfFiles, 8));
DataOut^[2] := WORD_TO_BYTE(NvDataIn^.wNumberOfFiles);

DataOut^[3] := WORD_TO_BYTE(SHR(NvDataIn^.wSelectedFile, 8));
DataOut^[4] := WORD_TO_BYTE(NvDataIn^.wSelectedFile);

DataOut^[5] := NvDataIn^.abAdr[0];
DataOut^[6] := NvDataIn^.abAdr[1];
DataOut^[7] := NvDataIn^.abAdr[2];
DataOut^[8] := NvDataIn^.abAdr[3];
DataOut^[9] := NvDataIn^.abAdr[4];
DataOut^[10] := NvDataIn^.abAdr[5];
DataOut^[11] := NvDataIn^.abAdr[6];
DataOut^[12] := NvDataIn^.abAdr[7];
DataOut^[13] := NvDataIn^.abAdr[8];
DataOut^[14] := NvDataIn^.abAdr[9];
DataOut^[15] := NvDataIn^.abAdr[10];
DataOut^[16] := NvDataIn^.abAdr[11];
DataOut^[17] := NvDataIn^.abAdr[12];
DataOut^[18] := NvDataIn^.abAdr[13];
DataOut^[19] := NvDataIn^.abAdr[14];
DataOut^[20] := NvDataIn^.abAdr[15];
DataOut^[21] := NvDataIn^.abAdr[16];
DataOut^[22] := NvDataIn^.abAdr[17];
DataOut^[23] := NvDataIn^.abAdr[18];
DataOut^[24] := NvDataIn^.abAdr[19];
DataOut^[25] := NvDataIn^.abAdr[20];
DataOut^[26] := NvDataIn^.abAdr[21];

FuSnvtFileStatusToRaw := TRUE;
END_FUNCTION

(* POU LON/Module_1/Internal/FuSendNviValueReq_Module_1, ST *)
FUNCTION FuSendNviValueReq_Module_1 : BOOL
(******************************************)
(* Automatic generated code, do not edit! *)
(******************************************)
VAR_INPUT
	ptInternalUseOnly : POINTER TO BYTE;
	bNvIndex : BYTE;
END_VAR
IF ptInternalUseOnly^.0 = TRUE THEN
	OutDataTelegram_Module_1[0] := C2M_NV_VALUE_QRY;
	OutDataTelegram_Module_1[1] := bNvIndex;

	mbxModule_1.bTxPrio := 1;
	mbxModule_1.bTxProtID := 0;
	mbxModule_1.pbTxData := ADR(OutDataTelegram_Module_1);
	mbxModule_1.unTxLen := 2;
	mbxModule_1.MBX_SEND();

	IF (mbxModule_1.nError <> MBX_OK) THEN
		FuSendNviValueReq_Module_1 := FALSE;
		RETURN;
	END_IF
	ptInternalUseOnly^.0 := FALSE;
END_IF

FuSendNviValueReq_Module_1 := TRUE;
END_FUNCTION

(* POU LON/Module_1/NV_Interface/Module_1_Virtualfunctionalblock, ST *)
FUNCTION_BLOCK Module_1_Virtualfunctionalblock
(******************************************)
(* Automatic generated code, do not edit! *)
(******************************************)
VAR_INPUT
	bObjectIndex : BYTE := 0;
	VT_TimeSet : typSnvtTimeStamp;
	VT_Request : typSnvtObjRequest;
	VT_AlarmSet : typSnvtAlarm;
	VT_DHW_ModeSet : typSnvtHvacMode;
	VT_DHW_SetPoint : typSnvtTempP;
	VT_CFD_SetEn : typSnvtSwitch;
	VT_CFD_SetMode : typSnvtHvacMode;
	VT_CFD_SetPoint : typSnvtTempP;

END_VAR
VAR_OUTPUT
	VT_Status : typSnvtObjStatus;
	VT_Alarm : typSnvtAlarm;
	VT_RlyState : typSnvtState;
	VT_DHW_ActTemp : typSnvtTempP;
	VT_DHW_SetTemp : typSnvtTempP;
	VT_CFD_GetEn : typSnvtSwitch;
	VT_CFD_Temp : typSnvtTempP;
	VT_CFD_SetTemp : typSnvtTempP;
	SNVT_casa : typSnvtAlarm;

END_VAR
VAR
	xSetOnce : BOOL := TRUE;
	xDataInUpdated : BOOL := FALSE;
	VT_TimeSetLast: typSnvtTimeStamp;
	VT_RequestLast: typSnvtObjRequest;
	VT_AlarmSetLast: typSnvtAlarm;
	VT_CFD_SetEnLast: typSnvtSwitch;
	paNviSnvtAlarm : ARRAY[0..1] OF POINTER TO typSnvtAlarm;
	aNviSnvtAlarmIndex : ARRAY[0..1] OF BYTE := 9,16;
	paNviSnvtTempP : ARRAY[0..3] OF POINTER TO typSnvtTempP;
	aNviSnvtTempPIndex : ARRAY[0..3] OF BYTE := 11,12,14,15;
	paNvoSnvtHvacMode : ARRAY[0..1] OF POINTER TO typSnvtHvacMode;
	aNvoSnvtHvacModeIndex : ARRAY[0..1] OF BYTE := 3,6;
	aNvoSnvtHvacModeLast : ARRAY[0..1] OF typSnvtHvacMode;
	aNvoSnvtHvacModePriority : ARRAY[0..0] OF BYTE := 16#00;
	paNvoSnvtTempP : ARRAY[0..1] OF POINTER TO typSnvtTempP;
	aNvoSnvtTempPIndex : ARRAY[0..1] OF BYTE := 4,7;
	aNvoSnvtTempPLast : ARRAY[0..1] OF typSnvtTempP;
	aNvoSnvtTempPPriority : ARRAY[0..0] OF BYTE := 16#00;

	cmd : BYTE;
	z : INT;
	bNvRelativeIdx : BYTE;
	bNvAbsoluteIdx : BYTE;
	wCpRelativeIdx : WORD;
	wCpAbsoluteIdx : WORD;
END_VAR
VAR CONSTANT
	bNvStartIndex : BYTE := 5;
	wCpStartIndex : WORD := 65535;
	bLmoCount : BYTE := 1;
END_VAR
IF (xInitRunning_Module_1 = TRUE) AND (xSetOnce = TRUE) THEN
	xSetOnce := FALSE;
	CachePointers();
	SetUpdateFlags();
END_IF

CheckUpdateFlags();
IF (xInitRunning_Module_1 = FALSE) AND (xDataInUpdated = FALSE) THEN
	IF (mbxModule_1.bStatus.0) THEN
		SendValueRequest();
	END_IF
END_IF

IF (xInitRunning_Module_1 = FALSE) AND (mbxModule_1.bStatus.0) THEN
	xSetOnce := TRUE;
	xDataInUpdated := FALSE;
	IF ((NOT FuMemCompare(ADR(VT_TimeSetLast), ADR(VT_TimeSet), ADR(VT_TimeSet.bStatusInformation) - ADR(VT_TimeSet))) OR (VT_TimeSet.bStatusInformation.7 = TRUE) OR (VT_TimeSetLast.bInternalUseOnly.1 = TRUE)) THEN
		FuSnvtTimeStampToRaw(ADR(VT_TimeSet), ADR(OutDataTelegram_Module_1[2]));

		bNvAbsoluteIdx := bNvStartIndex + bObjectIndex + (0 * bLmoCount);

		IF (FuDoNvoUpdate_Module_1(ADR(VT_TimeSet), ADR(VT_TimeSetLast), ADR(VT_TimeSet.bInternalUseOnly), ADR(VT_TimeSetLast.bInternalUseOnly), ADR(VT_TimeSet.bStatusInformation), bNvAbsoluteIdx, 7, SIZEOF(VT_TimeSet)) = FALSE) THEN
			RETURN;
		END_IF
	END_IF
	IF ((NOT FuMemCompare(ADR(VT_RequestLast), ADR(VT_Request), ADR(VT_Request.bStatusInformation) - ADR(VT_Request))) OR (VT_Request.bStatusInformation.7 = TRUE) OR (VT_RequestLast.bInternalUseOnly.1 = TRUE)) THEN
		FuSnvtObjRequestToRaw(ADR(VT_Request), ADR(OutDataTelegram_Module_1[2]));

		bNvAbsoluteIdx := bNvStartIndex + bObjectIndex + (1 * bLmoCount);

		IF (FuDoNvoUpdate_Module_1(ADR(VT_Request), ADR(VT_RequestLast), ADR(VT_Request.bInternalUseOnly), ADR(VT_RequestLast.bInternalUseOnly), ADR(VT_Request.bStatusInformation), bNvAbsoluteIdx, 3, SIZEOF(VT_Request)) = FALSE) THEN
			RETURN;
		END_IF
	END_IF
	IF ((NOT FuMemCompare(ADR(VT_AlarmSetLast), ADR(VT_AlarmSet), ADR(VT_AlarmSet.bStatusInformation) - ADR(VT_AlarmSet))) OR (VT_AlarmSet.bStatusInformation.7 = TRUE) OR (VT_AlarmSetLast.bInternalUseOnly.1 = TRUE)) THEN
		FuSnvtAlarmToRaw(ADR(VT_AlarmSet), ADR(OutDataTelegram_Module_1[2]));

		bNvAbsoluteIdx := bNvStartIndex + bObjectIndex + (2 * bLmoCount);

		IF (FuDoNvoUpdate_Module_1(ADR(VT_AlarmSet), ADR(VT_AlarmSetLast), ADR(VT_AlarmSet.bInternalUseOnly), ADR(VT_AlarmSetLast.bInternalUseOnly), ADR(VT_AlarmSet.bStatusInformation), bNvAbsoluteIdx, 29, SIZEOF(VT_AlarmSet)) = FALSE) THEN
			RETURN;
		END_IF
	END_IF
	IF ((NOT FuMemCompare(ADR(VT_CFD_SetEnLast), ADR(VT_CFD_SetEn), ADR(VT_CFD_SetEn.bStatusInformation) - ADR(VT_CFD_SetEn))) OR (VT_CFD_SetEn.bStatusInformation.7 = TRUE) OR (VT_CFD_SetEnLast.bInternalUseOnly.1 = TRUE)) THEN
		FuSnvtSwitchToRaw(ADR(VT_CFD_SetEn), ADR(OutDataTelegram_Module_1[2]));

		bNvAbsoluteIdx := bNvStartIndex + bObjectIndex + (5 * bLmoCount);

		IF (FuDoNvoUpdate_Module_1(ADR(VT_CFD_SetEn), ADR(VT_CFD_SetEnLast), ADR(VT_CFD_SetEn.bInternalUseOnly), ADR(VT_CFD_SetEnLast.bInternalUseOnly), ADR(VT_CFD_SetEn.bStatusInformation), bNvAbsoluteIdx, 2, SIZEOF(VT_CFD_SetEn)) = FALSE) THEN
			RETURN;
		END_IF
	END_IF
	FOR z := 0 TO 1 DO
		IF ((NOT FuMemCompare(ADR(aNvoSnvtHvacModeLast[z]), paNvoSnvtHvacMode[z], ADR(paNvoSnvtHvacMode[z]^.bStatusInformation) - paNvoSnvtHvacMode[z])) OR (paNvoSnvtHvacMode[z]^.bStatusInformation.7 = TRUE) OR (aNvoSnvtHvacModeLast[z].bInternalUseOnly.1 = TRUE)) THEN
			FuSnvtHvacModeToRaw(paNvoSnvtHvacMode[z], ADR(OutDataTelegram_Module_1[2]));

			bNvAbsoluteIdx := bNvStartIndex + bObjectIndex + (aNvoSnvtHvacModeIndex[z] * bLmoCount);

			IF (FuDoNvoUpdate_Module_1(paNvoSnvtHvacMode[z], ADR(aNvoSnvtHvacModeLast[z]), ADR(paNvoSnvtHvacMode[z]^.bInternalUseOnly), ADR(aNvoSnvtHvacModeLast[z].bInternalUseOnly), ADR(paNvoSnvtHvacMode[z]^.bStatusInformation), bNvAbsoluteIdx, 1, SIZEOF(aNvoSnvtHvacModeLast[z])) = FALSE) THEN
				RETURN;
			END_IF
		END_IF
	END_FOR
	FOR z := 0 TO 1 DO
		IF ((NOT FuMemCompare(ADR(aNvoSnvtTempPLast[z]), paNvoSnvtTempP[z], ADR(paNvoSnvtTempP[z]^.bStatusInformation) - paNvoSnvtTempP[z])) OR (paNvoSnvtTempP[z]^.bStatusInformation.7 = TRUE) OR (aNvoSnvtTempPLast[z].bInternalUseOnly.1 = TRUE)) THEN
			FuSnvtTempPToRaw(paNvoSnvtTempP[z], ADR(OutDataTelegram_Module_1[2]));

			bNvAbsoluteIdx := bNvStartIndex + bObjectIndex + (aNvoSnvtTempPIndex[z] * bLmoCount);

			IF (FuDoNvoUpdate_Module_1(paNvoSnvtTempP[z], ADR(aNvoSnvtTempPLast[z]), ADR(paNvoSnvtTempP[z]^.bInternalUseOnly), ADR(aNvoSnvtTempPLast[z].bInternalUseOnly), ADR(paNvoSnvtTempP[z]^.bStatusInformation), bNvAbsoluteIdx, 2, SIZEOF(aNvoSnvtTempPLast[z])) = FALSE) THEN
				RETURN;
			END_IF
		END_IF
	END_FOR

END_IF
END_FUNCTION_BLOCK
ACTION CachePointers:
paNviSnvtAlarm[0] := ADR(VT_Alarm);
paNviSnvtAlarm[1] := ADR(SNVT_casa);
paNviSnvtTempP[0] := ADR(VT_DHW_ActTemp);
paNviSnvtTempP[1] := ADR(VT_DHW_SetTemp);
paNviSnvtTempP[2] := ADR(VT_CFD_Temp);
paNviSnvtTempP[3] := ADR(VT_CFD_SetTemp);
paNvoSnvtHvacMode[0] := ADR(VT_DHW_ModeSet);
paNvoSnvtHvacMode[1] := ADR(VT_CFD_SetMode);
paNvoSnvtTempP[0] := ADR(VT_DHW_SetPoint);
paNvoSnvtTempP[1] := ADR(VT_CFD_SetPoint);
;
END_ACTION
ACTION CheckUpdateFlags:
xDataInUpdated := (NOT VT_Status.bInternalUseOnly.0) AND (NOT VT_RlyState.bInternalUseOnly.0) AND (NOT VT_CFD_GetEn.bInternalUseOnly.0) AND TRUE;
FOR z := 0 TO 1 DO
	xDataInUpdated := xDataInUpdated AND (NOT paNviSnvtAlarm[z]^.bInternalUseOnly.0);
END_FOR
FOR z := 0 TO 3 DO
	xDataInUpdated := xDataInUpdated AND (NOT paNviSnvtTempP[z]^.bInternalUseOnly.0);
END_FOR
END_ACTION
ACTION DataReceived:
cmd := InDataTelegram_Module_1[0];
IF (cmd = M2C_NVI_UPDT_OCCD) OR (cmd = M2C_NV_VALUE_RSP) OR (cmd = M2C_NVI_UPDT_TOUT) THEN
	bNvRelativeIdx := (InDataTelegram_Module_1[1] - bNvStartIndex - bObjectIndex) / bLmoCount;
	CASE bNvRelativeIdx OF
	8:
		IF (cmd = M2C_NVI_UPDT_OCCD) OR (cmd = M2C_NV_VALUE_RSP) THEN
			IF (unLastLen_mbxModule_1 = (2 + 6)) THEN
				FuRawToSnvtObjStatus(ADR(InDataTelegram_Module_1[2]), ADR(VT_Status));
				VT_Status.bInternalUseOnly.0 := FALSE;
				VT_Status.bStatusInformation := FuInkrementNviStatus(VT_Status.bStatusInformation);
			ELSIF (unLastLen_mbxModule_1 = 2) THEN
				VT_Status.bStatusInformation := FuInkrementNviStatus(VT_Status.bStatusInformation);
			END_IF
		ELSIF (cmd = M2C_NVI_UPDT_TOUT) THEN
			IF (unLastLen_mbxModule_1 = 3) THEN
				VT_Status.bStatusInformation.4 := BYTE_TO_BOOL(InDataTelegram_Module_1[2]);
			END_IF
		END_IF
	10:
		IF (cmd = M2C_NVI_UPDT_OCCD) OR (cmd = M2C_NV_VALUE_RSP) THEN
			IF (unLastLen_mbxModule_1 = (2 + 2)) THEN
				FuRawToSnvtState(ADR(InDataTelegram_Module_1[2]), ADR(VT_RlyState));
				VT_RlyState.bInternalUseOnly.0 := FALSE;
				VT_RlyState.bStatusInformation := FuInkrementNviStatus(VT_RlyState.bStatusInformation);
			ELSIF (unLastLen_mbxModule_1 = 2) THEN
				VT_RlyState.bStatusInformation := FuInkrementNviStatus(VT_RlyState.bStatusInformation);
			END_IF
		ELSIF (cmd = M2C_NVI_UPDT_TOUT) THEN
			IF (unLastLen_mbxModule_1 = 3) THEN
				VT_RlyState.bStatusInformation.4 := BYTE_TO_BOOL(InDataTelegram_Module_1[2]);
			END_IF
		END_IF
	13:
		IF (cmd = M2C_NVI_UPDT_OCCD) OR (cmd = M2C_NV_VALUE_RSP) THEN
			IF (unLastLen_mbxModule_1 = (2 + 2)) THEN
				FuRawToSnvtSwitch(ADR(InDataTelegram_Module_1[2]), ADR(VT_CFD_GetEn));
				VT_CFD_GetEn.bInternalUseOnly.0 := FALSE;
				VT_CFD_GetEn.bStatusInformation := FuInkrementNviStatus(VT_CFD_GetEn.bStatusInformation);
			ELSIF (unLastLen_mbxModule_1 = 2) THEN
				VT_CFD_GetEn.bStatusInformation := FuInkrementNviStatus(VT_CFD_GetEn.bStatusInformation);
			END_IF
		ELSIF (cmd = M2C_NVI_UPDT_TOUT) THEN
			IF (unLastLen_mbxModule_1 = 3) THEN
				VT_CFD_GetEn.bStatusInformation.4 := BYTE_TO_BOOL(InDataTelegram_Module_1[2]);
			END_IF
		END_IF
	9, 16:
		IF (cmd = M2C_NVI_UPDT_OCCD) OR (cmd = M2C_NV_VALUE_RSP) THEN
			IF (unLastLen_mbxModule_1 = (2 + 29)) THEN
				FOR z := 0 TO 1 DO
					IF aNviSnvtAlarmIndex[z] = bNvRelativeIdx THEN
						FuRawToSnvtAlarm(ADR(InDataTelegram_Module_1[2]), paNviSnvtAlarm[z]);
						paNviSnvtAlarm[z]^.bInternalUseOnly.0 := FALSE;
						paNviSnvtAlarm[z]^.bStatusInformation := FuInkrementNviStatus(paNviSnvtAlarm[z]^.bStatusInformation);
						EXIT;
					END_IF
				END_FOR
			ELSIF (unLastLen_mbxModule_1 = 2) THEN
				FOR z := 0 TO 1 DO
					IF aNviSnvtAlarmIndex[z] = bNvRelativeIdx THEN
						paNviSnvtAlarm[z]^.bStatusInformation := FuInkrementNviStatus(paNviSnvtAlarm[z]^.bStatusInformation);
						EXIT;
					END_IF
				END_FOR
			END_IF
		ELSIF (cmd = M2C_NVI_UPDT_TOUT) THEN
			IF (unLastLen_mbxModule_1 = 3) THEN
				FOR z := 0 TO 1 DO
					IF aNviSnvtAlarmIndex[z] = bNvRelativeIdx THEN
						paNviSnvtAlarm[z]^.bStatusInformation.4 := BYTE_TO_BOOL(InDataTelegram_Module_1[2]);
						EXIT;
					END_IF
				END_FOR
			END_IF
		END_IF
	11..12, 14..15:
		IF (cmd = M2C_NVI_UPDT_OCCD) OR (cmd = M2C_NV_VALUE_RSP) THEN
			IF (unLastLen_mbxModule_1 = (2 + 2)) THEN
				FOR z := 0 TO 3 DO
					IF aNviSnvtTempPIndex[z] = bNvRelativeIdx THEN
						FuRawToSnvtTempP(ADR(InDataTelegram_Module_1[2]), paNviSnvtTempP[z]);
						paNviSnvtTempP[z]^.bInternalUseOnly.0 := FALSE;
						paNviSnvtTempP[z]^.bStatusInformation := FuInkrementNviStatus(paNviSnvtTempP[z]^.bStatusInformation);
						EXIT;
					END_IF
				END_FOR
			ELSIF (unLastLen_mbxModule_1 = 2) THEN
				FOR z := 0 TO 3 DO
					IF aNviSnvtTempPIndex[z] = bNvRelativeIdx THEN
						paNviSnvtTempP[z]^.bStatusInformation := FuInkrementNviStatus(paNviSnvtTempP[z]^.bStatusInformation);
						EXIT;
					END_IF
				END_FOR
			END_IF
		ELSIF (cmd = M2C_NVI_UPDT_TOUT) THEN
			IF (unLastLen_mbxModule_1 = 3) THEN
				FOR z := 0 TO 3 DO
					IF aNviSnvtTempPIndex[z] = bNvRelativeIdx THEN
						paNviSnvtTempP[z]^.bStatusInformation.4 := BYTE_TO_BOOL(InDataTelegram_Module_1[2]);
						EXIT;
					END_IF
				END_FOR
			END_IF
		END_IF

	END_CASE
ELSIF (cmd = M2C_CP_VALUE_RSP) THEN
	wCpRelativeIdx := ((InDataTelegram_Module_1[1] + InDataTelegram_Module_1[2] * 256) - wCpStartIndex - bObjectIndex) / bLmoCount;
	CASE wCpRelativeIdx OF

	END_CASE
END_IF
END_ACTION
ACTION ResetNviUpdate:
VT_Status.bStatusInformation := VT_Status.bStatusInformation AND 16#F8;
VT_RlyState.bStatusInformation := VT_RlyState.bStatusInformation AND 16#F8;
VT_CFD_GetEn.bStatusInformation := VT_CFD_GetEn.bStatusInformation AND 16#F8;
FOR z := 0 TO 1 DO
	paNviSnvtAlarm[z]^.bStatusInformation := paNviSnvtAlarm[z]^.bStatusInformation AND 16#F8;
END_FOR
FOR z := 0 TO 3 DO
	paNviSnvtTempP[z]^.bStatusInformation := paNviSnvtTempP[z]^.bStatusInformation AND 16#F8;
END_FOR
;
END_ACTION
ACTION SendValueRequest:
IF (FuSendNviValueReq_Module_1(ADR(VT_Status.bInternalUseOnly), bNvStartIndex + bObjectIndex + (8 * bLmoCount)) = FALSE) THEN
	RETURN;
END_IF

IF (FuSendNviValueReq_Module_1(ADR(VT_RlyState.bInternalUseOnly), bNvStartIndex + bObjectIndex + (10 * bLmoCount)) = FALSE) THEN
	RETURN;
END_IF

IF (FuSendNviValueReq_Module_1(ADR(VT_CFD_GetEn.bInternalUseOnly), bNvStartIndex + bObjectIndex + (13 * bLmoCount)) = FALSE) THEN
	RETURN;
END_IF

FOR z := 0 TO 1 DO
	IF (FuSendNviValueReq_Module_1(ADR(paNviSnvtAlarm[z]^.bInternalUseOnly), bNvStartIndex + bObjectIndex + (aNviSnvtAlarmIndex[z] * bLmoCount)) = FALSE) THEN
		RETURN;
	END_IF;
END_FOR;
FOR z := 0 TO 3 DO
	IF (FuSendNviValueReq_Module_1(ADR(paNviSnvtTempP[z]^.bInternalUseOnly), bNvStartIndex + bObjectIndex + (aNviSnvtTempPIndex[z] * bLmoCount)) = FALSE) THEN
		RETURN;
	END_IF;
END_FOR;
;
END_ACTION
ACTION SetUpdateFlags:
VT_TimeSetLast.bInternaluseOnly.1 := TRUE;
VT_TimeSetLast.bInternaluseOnly.7 := FALSE;
VT_RequestLast.bInternaluseOnly.1 := TRUE;
VT_RequestLast.bInternaluseOnly.7 := FALSE;
VT_AlarmSetLast.bInternaluseOnly.1 := TRUE;
VT_AlarmSetLast.bInternaluseOnly.7 := FALSE;
VT_CFD_SetEnLast.bInternaluseOnly.1 := TRUE;
VT_CFD_SetEnLast.bInternaluseOnly.7 := FALSE;
VT_Status.bInternaluseOnly.0 := TRUE;
VT_RlyState.bInternaluseOnly.0 := TRUE;
VT_CFD_GetEn.bInternaluseOnly.0 := TRUE;
FOR z := 0 TO 1 DO
	paNviSnvtAlarm[z]^.bInternaluseOnly.0 := TRUE;
END_FOR;
FOR z := 0 TO 3 DO
	paNviSnvtTempP[z]^.bInternaluseOnly.0 := TRUE;
END_FOR;
FOR z := 0 TO 1 DO
	aNvoSnvtHvacModeLast[z].bInternaluseOnly.1 := TRUE;
	aNvoSnvtHvacModeLast[z].bInternaluseOnly.7 := (SHR(aNvoSnvtHvacModePriority[z / 8], z MOD 8) AND 1) <> 0;
END_FOR;
FOR z := 0 TO 1 DO
	aNvoSnvtTempPLast[z].bInternaluseOnly.1 := TRUE;
	aNvoSnvtTempPLast[z].bInternaluseOnly.7 := (SHR(aNvoSnvtTempPPriority[z / 8], z MOD 8) AND 1) <> 0;
END_FOR;
;
END_ACTION

(* POU LON/Shared/Internal/FuSnvtTimeStampToRaw, ST *)
FUNCTION FuSnvtTimeStampToRaw : BOOL
(******************************************)
(* Automatic generated code, do not edit! *)
(******************************************)
VAR_INPUT
	NvDataIn :  POINTER TO typSnvtTimeStamp;
	DataOut : POINTER TO ARRAY[0..6] OF BYTE;
END_VAR
VAR
END_VAR
DataOut^[0] := INT_TO_BYTE(SHR(NvDataIn^.iYear, 8));
DataOut^[1] := INT_TO_BYTE(NvDataIn^.iYear);

DataOut^[2] := NvDataIn^.bMonth;

DataOut^[3] := NvDataIn^.bDay;

DataOut^[4] := NvDataIn^.bHour;

DataOut^[5] := NvDataIn^.bMinute;

DataOut^[6] := NvDataIn^.bSecond;

FuSnvtTimeStampToRaw := TRUE;
END_FUNCTION

(* POU LON/Shared/Internal/FuSnvtObjRequestToRaw, ST *)
FUNCTION FuSnvtObjRequestToRaw : BOOL
(******************************************)
(* Automatic generated code, do not edit! *)
(******************************************)
VAR_INPUT
	NvDataIn :  POINTER TO typSnvtObjRequest;
	DataOut : POINTER TO ARRAY[0..2] OF BYTE;
END_VAR
VAR
END_VAR
DataOut^[0] := WORD_TO_BYTE(SHR(NvDataIn^.wObjectId, 8));
DataOut^[1] := WORD_TO_BYTE(NvDataIn^.wObjectId);

DataOut^[2] := NvDataIn^.bObjectRequest;

FuSnvtObjRequestToRaw := TRUE;
END_FUNCTION

(* POU LON/Shared/Internal/FuSnvtAlarmToRaw, ST *)
FUNCTION FuSnvtAlarmToRaw : BOOL
(******************************************)
(* Automatic generated code, do not edit! *)
(******************************************)
VAR_INPUT
	NvDataIn :  POINTER TO typSnvtAlarm;
	DataOut : POINTER TO ARRAY[0..28] OF BYTE;
END_VAR
VAR
END_VAR
DataOut^[0] := NvDataIn^.abLocation[0];
DataOut^[1] := NvDataIn^.abLocation[1];
DataOut^[2] := NvDataIn^.abLocation[2];
DataOut^[3] := NvDataIn^.abLocation[3];
DataOut^[4] := NvDataIn^.abLocation[4];
DataOut^[5] := NvDataIn^.abLocation[5];

DataOut^[6] := WORD_TO_BYTE(SHR(NvDataIn^.wObjectId, 8));
DataOut^[7] := WORD_TO_BYTE(NvDataIn^.wObjectId);

DataOut^[8] := NvDataIn^.bAlarmType;

DataOut^[9] := NvDataIn^.bPriorityLevel;

DataOut^[10] := WORD_TO_BYTE(SHR(NvDataIn^.wIndexToSnvt, 8));
DataOut^[11] := WORD_TO_BYTE(NvDataIn^.wIndexToSnvt);

DataOut^[12] := NvDataIn^.abValue[0];
DataOut^[13] := NvDataIn^.abValue[1];
DataOut^[14] := NvDataIn^.abValue[2];
DataOut^[15] := NvDataIn^.abValue[3];

DataOut^[16] := WORD_TO_BYTE(SHR(NvDataIn^.wYear, 8));
DataOut^[17] := WORD_TO_BYTE(NvDataIn^.wYear);

DataOut^[18] := NvDataIn^.bMonth;

DataOut^[19] := NvDataIn^.bDay;

DataOut^[20] := NvDataIn^.bHour;

DataOut^[21] := NvDataIn^.bMinute;

DataOut^[22] := NvDataIn^.bSecond;

DataOut^[23] := WORD_TO_BYTE(SHR(NvDataIn^.wMillisecond, 8));
DataOut^[24] := WORD_TO_BYTE(NvDataIn^.wMillisecond);

DataOut^[25] := NvDataIn^.abAlarmLimit[0];
DataOut^[26] := NvDataIn^.abAlarmLimit[1];
DataOut^[27] := NvDataIn^.abAlarmLimit[2];
DataOut^[28] := NvDataIn^.abAlarmLimit[3];

FuSnvtAlarmToRaw := TRUE;
END_FUNCTION

(* POU LON/Shared/Internal/FuSnvtSwitchToRaw, ST *)
FUNCTION FuSnvtSwitchToRaw : BOOL
(******************************************)
(* Automatic generated code, do not edit! *)
(******************************************)
VAR_INPUT
	NvDataIn :  POINTER TO typSnvtSwitch;
	DataOut : POINTER TO ARRAY[0..1] OF BYTE;
END_VAR
VAR
END_VAR
DataOut^[0] := NvDataIn^.bValue;

DataOut^[1] := NvDataIn^.siState;

FuSnvtSwitchToRaw := TRUE;
END_FUNCTION

(* POU LON/Shared/Internal/FuSnvtHvacModeToRaw, ST *)
FUNCTION FuSnvtHvacModeToRaw : BOOL
(******************************************)
(* Automatic generated code, do not edit! *)
(******************************************)
VAR_INPUT
	NvDataIn :  POINTER TO typSnvtHvacMode;
	DataOut : POINTER TO ARRAY[0..0] OF BYTE;
END_VAR
VAR
END_VAR
DataOut^[0] := NvDataIn^.bSnvtHvacMode;

FuSnvtHvacModeToRaw := TRUE;
END_FUNCTION

(* POU LON/Shared/Internal/FuSnvtTempPToRaw, ST *)
FUNCTION FuSnvtTempPToRaw : BOOL
(******************************************)
(* Automatic generated code, do not edit! *)
(******************************************)
VAR_INPUT
	NvDataIn :  POINTER TO typSnvtTempP;
	DataOut : POINTER TO ARRAY[0..1] OF BYTE;
END_VAR
VAR
END_VAR
DataOut^[0] := INT_TO_BYTE(SHR(NvDataIn^.iSnvtTempP, 8));
DataOut^[1] := INT_TO_BYTE(NvDataIn^.iSnvtTempP);

FuSnvtTempPToRaw := TRUE;
END_FUNCTION

(* POU TCP_Logger/Logger_Proc, ST *)
PROGRAM Logger_Proc
VAR
	c1:         	TCPCLIENT;
(*	c1:         	TCP_CLIENT; *)

	Open:	    	BOOL;
	IpAddr:			DWORD;
	InetAddr:		DWORD;
	Connected:  	BOOL;
	Error:      	DINT;
	TxTrig:     	BOOL;
	RxData:			ARRAY [0..MAX_RECEIVE_TCP_CLIENT] OF BYTE;
	RxLen:			DINT;

	Retry:			BYTE;	(* Counter for connection retries *)
	Recovered:		BYTE;	(* Counter for recovered unsent messages *)

	i:				DINT;
	pos:			DWORD;
	hFile:			DWORD;

	Str_HTTP_Response:STRING;



	Counter: INT;
END_VAR
(*=== State machine ===*)
CASE Logger.Status OF

	S_Logger_UNKNOWN:
		(* Startup *)
		Logger.SendReq:=FALSE;
		Open:=FALSE;
		Logger.Status:=S_Logger_IDLE;

	S_Logger_IDLE:
		(* Wait request *)
		IF Logger.SendReq THEN
			(* Resolve server name or use static IP *)
			IF LEN(Logger_SERVER)=0 THEN
				InetAddr:=SysSockInetAddr(Logger_IP);
			ELSE
				IpAddr:=SysSockGetHostByName(ADR(Logger_SERVER));
				DWORDSWAP(pIn:=ADR(IpAddr), pOut:=ADR(InetAddr));
			END_IF
			TxTrig:=FALSE;
			RxLen:=0;
			(* Open connection *)
			Open:=TRUE;
			Logger.Status:=S_Logger_WAITCONN;
		END_IF

	S_Logger_WAITCONN:
		(* Wait connection *)
		IF Connected THEN
			(* Send data *)
			TxTrig:=TRUE;
			Logger.Status:=S_Logger_WAITTX;
			Str_HTTP_Response:='';

		END_IF
		IF Error>0 THEN
			Open:=FALSE;
			Logger.Status:=S_Logger_ERROR;
		END_IF

	S_Logger_WAITTX:
		(* Wait transmission *)
		IF NOT TxTrig THEN
			Logger.Status:=S_Logger_WAITRESP;
		END_IF
		IF Error>0 THEN
			Open:=FALSE;
			Logger.Status:=S_Logger_ERROR;
		END_IF

	S_Logger_WAITRESP:
		(* Wait response *)
		IF Connected=FALSE (* OR TIMEOUT!! *) THEN
			Open:=FALSE;
			(* Check response *)
			IF RxLen>=4 AND CHKSTRING(pString:=ADR(RxData), pPattern:=ADR(Logger_CHECK)) THEN
				Logger.SendReq:=FALSE;
				Retry:=0;
				(* Check unsent messages to flush *)
				IF Recovered<Logger_RecoverMsgs THEN
					MsgChk();
					IF Logger.SendReq=TRUE THEN
						Recovered:=Recovered+1;
					ELSE
						Recovered:=0;
					END_IF
				ELSE
					Recovered:=0;
				END_IF
				Logger.Status:=S_Logger_IDLE;
			ELSE
				Logger.Status:=S_Logger_ERROR;
			END_IF
		END_IF

	S_Logger_ERROR:
		(* Connection error or send failure *)
		Retry:=Retry+1;
		IF Retry>Logger_ConnRetries THEN
			(* Save message as unsent *)
			MsgSave();
			Logger.SendReq:=FALSE;
			Retry:=0;
		END_IF
		Logger.Status:=S_Logger_IDLE;

ELSE
	Logger.Status:=S_Logger_UNKNOWN;
END_CASE



(*=== Execute client lib ===*)
c1(
	xOpenConnection			:= Open,
	dwInetAddr 				:= InetAddr,
	wPortNumber				:= Logger_PORT,
	ptSendData				:= ADR(Logger.SendData),
	diSendCount				:= Logger.SendLen,
	tConnectWatchdogTime	:= t#10s,
	xStartSend				:= TxTrig,
	aReceiveBuffer			:= RxData,
	diReceiveCount			:= RxLen,
	xConnected				=> Connected,
	diError					=> Error
);

(*

c1(
	xOpenConnection:= Open,
	sIPaddress:= Logger_IP,
	wPortNumber:= Logger_PORT,
	ptSendData:= ADR(Logger.SendData),
	diSendCount:= Logger.SendLen,
	xStartSend:= TxTrig,
	aReceiveBuffer:= RxData,
	diReceiveCount:= RxLen,
	xConnected=> Connected,
	diError=> Error);

		IF RxLen>0 THEN
			Str_HTTP_Response:='';
			FOR Counter:=0 TO 14 BY 1 DO
				Str_HTTP_Response:=CONCAT(Str_HTTP_Response, ASCIIBYTE_TO_STRING( RxData[Counter] ) );
			END_FOR;
		END_IF
*)


(*=== Process Rx data ===*)
(*IF RxLen>0 THEN
	RxLen:=0;
END_IF*)
END_PROGRAM
ACTION MsgChk:
(* Open index file *)
hFile:=SysFileOpen(Logger_IndexFile,'r');
IF hFile=0 THEN
	RETURN;
END_IF
(* Search oldest message to recover *)
SysFileSetPos(hFile,Logger.LastIdxPos);
Logger.SendLen:=0;
REPEAT
	SysFileRead(hFile, ADR(Logger.SendIdx), SIZEOF(Logger.SendIdx));
	pos:=SysFileGetPos(hFile);
	SysFileRead(hFile, ADR(Logger.SendLen), SIZEOF(Logger.SendLen));
UNTIL
	SysFileEOF(hFile) OR Logger.SendLen<>0
END_REPEAT
SysFileClose(hFile);
(* Delete index file when all messages are recovered *)
IF Logger.SendLen=0 THEN
	Logger.LastIdxPos:=0;
	SysFileDelete(Logger_IndexFile);
	RETURN;
END_IF
(* Recover message data *)
hFile:=SysFileOpen(Logger_DataFile,'r');
IF hFile<>0 THEN
	SysFileSetPos(hFile,Logger.SendIdx);
	SysFileRead(hFile,ADR(Logger.SendData),Logger.SendLen);
	Logger.SendReq:=TRUE;
	SysFileClose(hFile);
END_IF
(* Clear index entry *)
hFile:=SysFileOpen(Logger_IndexFile,'a');
IF hFile<>0 THEN
	SysFileSetPos(hFile,pos);
	i:=0;
	SysFileWrite(hFile, ADR(i), 4);
	Logger.LastIdxPos:=SysFileGetPos(hFile);
	SysFileClose(hFile);
END_IF
END_ACTION
ACTION MsgSave:
(* Add log position in recovery indexes *)
hFile:=SysFileOpen(Logger_IndexFile,'a');
SysFileWrite(hFile, ADR(Logger.SendIdx), SIZEOF(Logger.SendIdx));
SysFileWrite(hFile, ADR(Logger.SendLen), SIZEOF(Logger.SendLen));
SysFileClose(hFile);
END_ACTION

(* POU Utils Functions/TCPCLIENT, ST *)
FUNCTION_BLOCK TCPCLIENT
(***********************************************************************************************************	*)
(* Version: 1.3b                        			          													*)
(* Date: 28.10.2014                   				          							            			*)
(***********************************************************************************************************	*)
(* WAGO Kontakttechnik GmbH Hansastr. 27 32423 Minden(Westf.)													*)
(* Tel. +0049 571/887-0 Fax. +0049 571/887-0																	*)
(* Author: VB																									*)
(***********************************************************************************************************	*)
(*Description:	A TCP client to read and write data with additional connection watchdog							*)
(*History:																										*)
(*Version 1.3b: 28.10.2014: Use DWORD address for IP (Andrea Ravasio)											*)
(*Version 1.3: 11.02.2011: Changes according to 750-880/881											 			*)
(*Version 1.2: 29.08.2007 Bugfix TCP Client																		*)
(*Version 1.1: 15.01.2007 Changes according to FW11																*)
(*Version 1.0: 09.03.2006 Release																				*)
(***********************************************************************************************************	*)
VAR CONSTANT
	STATE_CREATE     				 : BYTE:= 0;
	STATE_OPEN     					 : BYTE:= 1;
	STATE_IOCTL    					 : BYTE:= 2;
	STATE_CONNECT     				 : BYTE:= 10;
	STATE_TX       					 : BYTE:= 20;
	STATE_RX       					 : BYTE:= 30;
	STATE_CLOSE    					 : BYTE:= 40;
	STATE_ERROR_TRAP			     : BYTE:= 200;
END_VAR

VAR_INPUT
	xOpenConnection					: BOOL;
	dwInetAddr						: DWORD; (* <== Use SysSockInetAddr() value or
													swapped bytes order of SysSockGetHostByName() value *)
	wPortNumber						: WORD;
	ptSendData						: POINTER TO ARRAY[0..MAX_SEND_TCP_CLIENT] OF BYTE;
	diSendCount						: DINT;
	tConnectWatchdogTime		    : TIME := t#10s;
END_VAR
VAR_OUTPUT
	xConnected						: BOOL;
	diError 						: DINT := 0;
END_VAR
(* ErrorCodes -----------------------------------------
	16#8001 => No socket descriptor available 
	16#8002 => SysSockSend returns -1 
	16#8003 => Socket was "gracefully closed" 
	16#8004 => switching to none blocking mode fails
	16#8005 => SysSockClose() returns FALSE 
    16#8006 => SysSockConnect() fails
    16#8007 => SysSockSend() fails
	16#8008 => error state machine 
	16#8009 => timeout while waiting for data from server 
------------------------------------------------------------*)
VAR_IN_OUT
	xStartSend							: BOOL;
	aReceiveBuffer						: ARRAY [0..MAX_RECEIVE_TCP_CLIENT] OF BYTE;
	diReceiveCount						: DINT;
END_VAR
VAR
	m_State								: BYTE := 0;
	m_ReceiveBuffer						: ARRAY [0..MAX_RECEIVE_TCP_CLIENT_SOCKET] OF BYTE;
	m_Socket							: DINT;
	m_AddressInfo						: SOCKADDRESS;
	m_BytesReceived						: DINT;
	m_diReturn							: DINT;
	m_xReturn							: BOOL;
	m_IoCtlParameter  					: DINT := 1; (* IOCTL-Parameter for non-blocking mode of sockets *)
	i									: INT;
	T_Connect							: TON;
	m_count								: DINT;
	diOption							: DINT := 1;
	m_Blocking   						: DINT := 0;
END_VAR
IF xOpenConnection THEN
	(* State maschine *)
	CASE  m_State OF

	(* -------------------------------------------------------------------------*)
	STATE_CREATE:
			(* create socket descriptor*)
			m_Socket := SysSockCreate(diAddressFamily	:= SOCKET_AF_INET,
													 diType		:= SOCKET_STREAM,
													 diProtocol := SOCKET_IPPROTO_TCP);
			IF m_Socket >= 0 THEN
			(*Set Push-Bit*)
				IF ADR(%MW0)=16#30000000  OR ADR(%MW0)=16#20000000 THEN (*841 or 881*)
					SysSockSetOption(
						diSocket:=m_Socket,
						diLevel:=6,
						diOption:=SOCKET_TCP_NODELAY,
						pOptionValue:=ADR(diOption),
						diOptionLength:=SIZEOF(diOption));
				ELSE
						;
				END_IF
				m_State := STATE_IOCTL; (* succesful *)
			ELSE
				diError := 16#8001;  (* no socket descriptor available *)
				m_State := STATE_ERROR_TRAP;
			END_IF

	(* -------------------------------------------------------------------------*)
	STATE_IOCTL: (* change  socket mode  to none blocking *)
		m_diReturn := SysSockIoctl( m_Socket, SOCKET_FIONBIO, ADR(m_IoCtlParameter));
		IF m_diReturn <> 0 THEN
			m_AddressInfo.sin_family := SOCKET_AF_INET;
			m_AddressInfo.sin_port := SysSockNtohs(wPortNumber);
			m_AddressInfo.sin_addr := dwInetAddr;
			m_State := STATE_CONNECT;
		ELSE
			diError := 16#8004;  (* switching to none blocking mode fails *)
			m_State := STATE_ERROR_TRAP;
		END_IF


	(* -------------------------------------------------------------------------*)
	STATE_CONNECT: (* connect with server *)
		T_Connect(IN:=TRUE , PT:=tConnectWatchdogTime);(*activate watchdog for establishing connection to a server*)
		m_xReturn := SysSockConnect ( m_Socket, ADR(m_AddressInfo),  SIZEOF(m_AddressInfo));
		IF m_xReturn THEN (* succesful *)
			IF xStartSend THEN
				m_State := STATE_TX;(*transmit data*)
			ELSE
				m_State := STATE_RX;(*wait for data from server*)
			END_IF
			xConnected:=TRUE;
			T_Connect(IN:=FALSE);
		ELSE
			IF T_Connect.Q THEN
				diError := 16#8006;  (* connect fails *)
				xConnected:=FALSE;
				T_Connect(IN:=FALSE);
				m_State := STATE_ERROR_TRAP;
				SysSockClose( m_Socket);
			ELSE
				m_State := STATE_CONNECT;(*client still  tries to set up connection*)
			END_IF
		END_IF


	STATE_TX:	 (* send TCP-message *)
		m_diReturn := SysSockSend(diSocket := m_Socket,
								  pbyBuffer := ADR(ptSendData^[0]),
								  diBufferSize := diSendCount-m_count,
								  diFlags := 0);

		CASE m_diReturn OF
		-1:	(* ERROR *)
			T_Connect(IN:=TRUE , PT:=CONNECT_WATCHDOG_TIME);(*activate watchdog to check communication*)
			IF t_Connect.Q THEN
				diError := 16#8007;
				T_Connect(IN:=FALSE);
				m_State:=STATE_CLOSE;
			END_IF
		0: (* socket was "gracefully closed" *)
			m_State := STATE_CLOSE;
			diError := 16#8003;
		ELSE (* succesful *)
			m_count:=m_count+m_diReturn;
			IF m_count>=diSendCount THEN
				diError := 16#0000;
				m_State := STATE_RX;
				m_count:=0;
				xStartSend:=FALSE;
			END_IF
			T_Connect(IN:=FALSE);
		END_CASE

	(* -------------------------------------------------------------------------*)
	STATE_RX: (* process receive data *)
			m_BytesReceived := SysSockRecv(	diSocket 	:= m_Socket,
										pbyBuffer 	:= ADR(m_ReceiveBuffer),		(* Address of receive buffer *)
										diBufferSize:= SIZEOF(m_ReceiveBuffer),
										diFlags		:= 0);

			CASE m_BytesReceived OF
			-1:	(* No data available or error occured *)
				T_Connect(IN:=TRUE , PT:=tConnectWatchdogTime);(*activate watchdog to check communication*)
				IF t_Connect.Q THEN
					diError:=16#8009;
					T_Connect(IN:=FALSE);
					m_State:=STATE_CLOSE;
				END_IF
				IF xStartSend THEN
					m_State:=STATE_TX	;(* WAIT IN THIS STATE  and check for arriving data or new send command*)
				END_IF;
			0: (* socket was "gracefully closed"  *)
				m_State:=STATE_CLOSE;
				diError := 16#8003;
			ELSE (* succesful *)
				diError := 16#0000;
				T_Connect(IN:=FALSE);
				(* Copy received data into receive buffer *)
				FOR i:= 0 TO DINT_TO_INT(m_BytesReceived	)-1 DO
					aReceiveBuffer[diReceiveCount]:= m_ReceiveBuffer[i];
					diReceiveCount:=(diReceiveCount+1) MOD SIZEOF(aReceiveBuffer);
				END_FOR

			END_CASE

	(* -------------------------------------------------------------------------*)
	STATE_CLOSE : (* close socket *)
		IF ADR(%MW0)=16#30000000  OR ADR(%MW0)=16#20000000 THEN (*841 or 881*)
			;
		ELSE
			SysSockShutdown(m_Socket, 0);;(*870*)
		END_IF
		m_xReturn := SysSockClose( m_Socket);
		m_Socket := -1;
		m_State := 0; (* succesful *)
		xConnected:=FALSE;
		T_Connect(IN:=FALSE);
	(* -------------------------------------------------------------------------*)
	STATE_ERROR_TRAP: (* error handling *)
		xConnected:=FALSE;

	ELSE  (* Bad FSM code trap  *)
			m_State:= STATE_ERROR_TRAP;
			diError:= 16#8008;
	END_CASE

ELSE(*close connection*)
	IF m_Socket >= 0 THEN
		IF ADR(%MW0)=16#30000000  OR ADR(%MW0)=16#20000000 THEN (*841 or 881*)
			;
		ELSE
			SysSockShutdown(m_Socket, 0);;(*870*)
		END_IF
		SysSockClose( m_Socket);
	END_IF
	m_Socket := -1;
	diError := 16#0000;
	m_State := STATE_CREATE;
	xConnected:=FALSE;
	T_Connect(IN:=FALSE);
END_IF
END_FUNCTION_BLOCK

(* POU Utils Functions/DWORDSWAP, ST *)
FUNCTION DWORDSWAP:BOOL
VAR_INPUT
	pIn:POINTER TO ARRAY[1..4] OF BYTE;
	pOut:POINTER TO ARRAY[1..4] OF BYTE;
END_VAR
VAR
END_VAR
pOut^[1]:=pIn^[4];
pOut^[2]:=pIn^[3];
pOut^[3]:=pIn^[2];
pOut^[4]:=pIn^[1];
END_FUNCTION

(* POU Utils Functions/CHKSTRING, ST *)
FUNCTION CHKSTRING : BOOL
VAR_INPUT
	pString: POINTER TO BYTE;
	pPattern: POINTER TO BYTE;
END_VAR
VAR
END_VAR
CHKSTRING:=TRUE;
WHILE pPattern^<>0 AND CHKSTRING DO
	IF pPattern^<>pString^ THEN CHKSTRING:=FALSE; END_IF
	pString:=pString+1;
	pPattern:=pPattern+1;
END_WHILE
END_FUNCTION

(* POU TCP_Remote/Remote_Proc, ST *)
PROGRAM Remote_Proc
VAR
	s1:         	TCPSERVER;
	Enable: 		BOOL;
	Connected: 		BOOL;
	Error: 			DINT;

	TxData:			ARRAY [0..MAX_SEND_TCP_SERVER] OF BYTE;
	TxLen:			DINT;
	TxTrig:			BOOL;

	RxData:			ARRAY [0..MAX_RECEIVE_TCP_SERVER] OF BYTE;
	RxLen:			DINT;

	Status:			DINT;

	(* Command interpreter *)

	Cmd_Buf:		ARRAY [0..MAX_RECEIVE_TCP_SERVER] OF BYTE;
	Cmd_Buf_U16:	POINTER TO WORD;
	Cmd_Buf_INT:	POINTER TO INT;
	Cmd_BufLen:		WORD;
	Cmd_St:			WORD;

	Cmd_Obj:		WORD;
	Cmd_ObjIdx:		WORD;
	Cmd_C:			WORD;
	Cmd_R:			WORD;
	Cmd_CLen:		WORD;
	Cmd_RLen:		WORD;

	i : WORD;
	j : INT;
	s2 : STRING;


		(* per aggiornare la data e l'ora *)
	SetAnno: INT;
	SetMese: INT;
	SetGiorno: INT;
	SetOra: INT;
	SetMinuti: INT;
	SetSecondi: INT;


END_VAR
(*=== State machine ===*)
CASE Status OF
	0: (* Startup *)
		TxLen:=0; TxTrig:=FALSE;
		RxLen:=0;
		Enable:=TRUE;
		Status:=1;

	1: (* Wait incoming connection *)
		IF Connected THEN
			(* Log access *)(*
			LogEv(EL_Log,EO_VPN,1,5,'Remote');*)
			(* Send welcome message *)(*
			ADDSTRING(pTxData:=ADR(TxData), pString:=ADR(Remote_WELCOME), TxLen:=TxLen);
			TxTrig:=TRUE;*)
			(* Reset vars *)
			Cmd_BufLen:=0;
			Cmd_St:=0;
			Status:=2;
		END_IF
		IF Error>1 THEN
			Enable:=FALSE;
			Status:=0;
		END_IF

